LIN {X 0,Y 584.047,Z 358.292,A -85,B 0,C 180,E1 26461.667,E2 26461.667} C_VEL
LIN {X 0,Y 584.039,Z 358.291,A -85,B 0,C 180,E1 26458.43,E2 26458.43} C_VEL
LIN {X 0,Y 584.051,Z 358.293,A -85,B 0,C 180,E1 26455.483,E2 26455.483} C_VEL
LIN {X 0,Y 584.043,Z 358.289,A -85,B 0,C 180,E1 26452.227,E2 26452.227} C_VEL
LIN {X 0,Y 584.062,Z 358.294,A -85,B 0,C 180,E1 26449.245,E2 26449.245} C_VEL
LIN {X 0,Y 584.1,Z 358.29,A -85,B 0,C 180,E1 26446.657,E2 26446.657} C_VEL
LIN {X 0,Y 583.09,Z 358.412,A -85,B 0,C 180,E1 26445.901,E2 26445.901} C_VEL
LIN {X 0,Y 576.621,Z 359.216,A -85,B 0,C 180,E1 26443.781,E2 26443.781} C_VEL
LIN {X 0,Y 576.114,Z 359.282,A -85,B 0,C 180,E1 26443.229,E2 26443.229} C_VEL
LIN {X 0,Y 576.112,Z 359.279,A -85,B 0,C 180,E1 26439.856,E2 26439.856} C_VEL
LIN {X 0,Y 576.152,Z 359.283,A -85,B 0,C 180,E1 26436.692,E2 26436.692} C_VEL
LIN {X 0,Y 576.109,Z 359.279,A -85,B 0,C 180,E1 26433.51,E2 26433.51} C_VEL
LIN {X 0,Y 576.163,Z 359.281,A -85,B 0,C 180,E1 26430.357,E2 26430.357} C_VEL
LIN {X 0,Y 576.11,Z 359.279,A -85,B 0,C 180,E1 26427.131,E2 26427.131} C_VEL
LIN {X 0,Y 576.16,Z 359.278,A -85,B 0,C 180,E1 26423.96,E2 26423.96} C_VEL
LIN {X 0,Y 576.115,Z 359.279,A -85,B 0,C 180,E1 26420.822,E2 26420.822} C_VEL
LIN {X 0,Y 576.152,Z 359.275,A -85,B 0,C 180,E1 26417.54,E2 26417.54} C_VEL
LIN {X 0,Y 576.133,Z 359.281,A -85,B 0,C 180,E1 26414.355,E2 26414.355} C_VEL
LIN {X 0,Y 576.129,Z 359.276,A -85,B 0,C 180,E1 26410.98,E2 26410.98} C_VEL
LIN {X 0,Y 576.156,Z 359.281,A -85,B 0,C 180,E1 26407.772,E2 26407.772} C_VEL
LIN {X 0,Y 576.125,Z 359.275,A -85,B 0,C 180,E1 26404.571,E2 26404.571} C_VEL
LIN {X 0,Y 576.154,Z 359.278,A -85,B 0,C 180,E1 26401.369,E2 26401.369} C_VEL
LIN {X 0,Y 576.129,Z 359.275,A -85,B 0,C 180,E1 26398.16,E2 26398.16} C_VEL
LIN {X 0,Y 576.155,Z 359.27,A -85,B 0,C 180,E1 26394.821,E2 26394.821} C_VEL
LIN {X 0,Y 576.16,Z 359.275,A -85,B 0,C 180,E1 26391.475,E2 26391.475} C_VEL
LIN {X 0,Y 576.135,Z 359.276,A -85,B 0,C 180,E1 26388.199,E2 26388.199} C_VEL
LIN {X 0,Y 576.149,Z 359.283,A -85,B 0,C 180,E1 26384.982,E2 26384.982} C_VEL
LIN {X 0,Y 576.161,Z 359.453,A -85,B 0,C 180,E1 26381.921,E2 26381.921} C_VEL
LIN {X 0,Y 577.208,Z 362.341,A -85,B 0,C 180,E1 26381.665,E2 26381.665} C_VEL
LIN {X 0,Y 582.648,Z 371.022,A -85,B 0,C 180,E1 26381.087,E2 26381.087} C_VEL
LIN {X 0,Y 581.66,Z 578.825,A -85,B 0,C 180,E1 26377.993,E2 26377.993} C_VEL
LIN {X 0,Y 581.046,Z 710.551,A -85,B 0,C 180,E1 26376.056,E2 26376.056} C_VEL
LIN {X 0,Y 580.715,Z 734.129,A -85,B 0,C 180,E1 26375.517,E2 26375.517} C_VEL
LIN {X 0,Y 580.401,Z 756.068,A -85,B 0,C 180,E1 26374.833,E2 26374.833} C_VEL
LIN {X 0,Y 579.918,Z 778.158,A -85,B 0,C 180,E1 26373.951,E2 26373.951} C_VEL
LIN {X 0,Y 579.481,Z 800.389,A -85,B 0,C 180,E1 26372.865,E2 26372.865} C_VEL
LIN {X 0,Y 578.947,Z 821.449,A -85,B 0,C 180,E1 26371.63,E2 26371.63} C_VEL
LIN {X 0,Y 578.423,Z 842.935,A -85,B 0,C 180,E1 26370.146,E2 26370.146} C_VEL
LIN {X 0,Y 577.968,Z 862.118,A -85,B 0,C 180,E1 26368.609,E2 26368.609} C_VEL
LIN {X 0,Y 577.481,Z 880.371,A -85,B 0,C 180,E1 26366.92,E2 26366.92} C_VEL
LIN {X 0,Y 577.086,Z 898.241,A -85,B 0,C 180,E1 26365.027,E2 26365.027} C_VEL
LIN {X 0,Y 576.768,Z 913.925,A -85,B 0,C 180,E1 26363.127,E2 26363.127} C_VEL
LIN {X 0,Y 576.482,Z 927.611,A -85,B 0,C 180,E1 26361.218,E2 26361.218} C_VEL
LIN {X 0,Y 576.279,Z 940.902,A -85,B 0,C 180,E1 26359.096,E2 26359.096} C_VEL
LIN {X 0,Y 576.134,Z 951.802,A -85,B 0,C 180,E1 26357.061,E2 26357.061} C_VEL
LIN {X 0,Y 576.034,Z 962.063,A -85,B 0,C 180,E1 26354.803,E2 26354.803} C_VEL
LIN {X 0,Y 575.951,Z 969.516,A -85,B 0,C 180,E1 26352.833,E2 26352.833} C_VEL
LIN {X 0,Y 575.908,Z 976.629,A -85,B 0,C 180,E1 26350.516,E2 26350.516} C_VEL
LIN {X 0,Y 575.923,Z 981.54,A -85,B 0,C 180,E1 26348.402,E2 26348.402} C_VEL
LIN {X 0,Y 575.899,Z 985.41,A -85,B 0,C 180,E1 26346.027,E2 26346.027} C_VEL
LIN {X 0,Y 575.883,Z 987.332,A -85,B 0,C 180,E1 26343.941,E2 26343.941} C_VEL
LIN {X 0,Y 575.901,Z 987.929,A -85,B 0,C 180,E1 26341.592,E2 26341.592} C_VEL
LIN {X 0,Y 575.91,Z 986.963,A -85,B 0,C 180,E1 26339.421,E2 26339.421} C_VEL
LIN {X 0,Y 575.903,Z 984.298,A -85,B 0,C 180,E1 26337.081,E2 26337.081} C_VEL
LIN {X 0,Y 575.926,Z 980.083,A -85,B 0,C 180,E1 26334.802,E2 26334.802} C_VEL
LIN {X 0,Y 575.937,Z 973.943,A -85,B 0,C 180,E1 26332.455,E2 26332.455} C_VEL
LIN {X 0,Y 576.001,Z 967.203,A -85,B 0,C 180,E1 26330.42,E2 26330.42} C_VEL
LIN {X 0,Y 576.072,Z 958.165,A -85,B 0,C 180,E1 26328.201,E2 26328.201} C_VEL
LIN {X 0,Y 576.199,Z 947.718,A -85,B 0,C 180,E1 26326.042,E2 26326.042} C_VEL
LIN {X 0,Y 576.354,Z 935.657,A -85,B 0,C 180,E1 26323.942,E2 26323.942} C_VEL
LIN {X 0,Y 576.619,Z 922.062,A -85,B 0,C 180,E1 26321.882,E2 26321.882} C_VEL
LIN {X 0,Y 576.933,Z 906.451,A -85,B 0,C 180,E1 26319.846,E2 26319.846} C_VEL
LIN {X 0,Y 577.278,Z 889.678,A -85,B 0,C 180,E1 26317.943,E2 26317.943} C_VEL
LIN {X 0,Y 577.706,Z 871.832,A -85,B 0,C 180,E1 26316.17,E2 26316.17} C_VEL
LIN {X 0,Y 578.182,Z 853.165,A -85,B 0,C 180,E1 26314.557,E2 26314.557} C_VEL
LIN {X 0,Y 578.662,Z 832.887,A -85,B 0,C 180,E1 26313.041,E2 26313.041} C_VEL
LIN {X 0,Y 579.219,Z 811.589,A -85,B 0,C 180,E1 26311.675,E2 26311.675} C_VEL
LIN {X 0,Y 579.672,Z 790.373,A -85,B 0,C 180,E1 26310.529,E2 26310.529} C_VEL
LIN {X 0,Y 580.158,Z 768.038,A -85,B 0,C 180,E1 26309.532,E2 26309.532} C_VEL
LIN {X 0,Y 580.516,Z 746.553,A -85,B 0,C 180,E1 26308.758,E2 26308.758} C_VEL
LIN {X 0,Y 580.89,Z 723.232,A -85,B 0,C 180,E1 26308.119,E2 26308.119} C_VEL
LIN {X 0,Y 581.099,Z 700.855,A -85,B 0,C 180,E1 26307.69,E2 26307.69} C_VEL
LIN {X 0,Y 582.078,Z 488.35,A -85,B 0,C 180,E1 26304.584,E2 26304.584} C_VEL
LIN {X 0,Y 582.542,Z 370.805,A -85,B 0,C 180,E1 26302.811,E2 26302.811} C_VEL
LIN {X 0,Y 576.646,Z 361.193,A -85,B 0,C 180,E1 26302.156,E2 26302.156} C_VEL
LIN {X 0,Y 576.178,Z 359.428,A -85,B 0,C 180,E1 26301.934,E2 26301.934} C_VEL
LIN {X 0,Y 576.126,Z 359.253,A -85,B 0,C 180,E1 26298.728,E2 26298.728} C_VEL
LIN {X 0,Y 576.152,Z 359.274,A -85,B 0,C 180,E1 26295.398,E2 26295.398} C_VEL
LIN {X 0,Y 576.155,Z 359.281,A -85,B 0,C 180,E1 26292.122,E2 26292.122} C_VEL
LIN {X 0,Y 576.139,Z 359.277,A -85,B 0,C 180,E1 26288.886,E2 26288.886} C_VEL
LIN {X 0,Y 576.143,Z 359.277,A -85,B 0,C 180,E1 26285.677,E2 26285.677} C_VEL
LIN {X 0,Y 576.148,Z 359.28,A -85,B 0,C 180,E1 26282.387,E2 26282.387} C_VEL
LIN {X 0,Y 576.156,Z 359.274,A -85,B 0,C 180,E1 26279.006,E2 26279.006} C_VEL
LIN {X 0,Y 576.138,Z 359.281,A -85,B 0,C 180,E1 26275.721,E2 26275.721} C_VEL
LIN {X 0,Y 576.153,Z 359.278,A -85,B 0,C 180,E1 26272.422,E2 26272.422} C_VEL
LIN {X 0,Y 576.123,Z 359.278,A -85,B 0,C 180,E1 26269.197,E2 26269.197} C_VEL
LIN {X 0,Y 576.159,Z 359.283,A -85,B 0,C 180,E1 26265.939,E2 26265.939} C_VEL
LIN {X 0,Y 576.139,Z 359.276,A -85,B 0,C 180,E1 26262.633,E2 26262.633} C_VEL
LIN {X 0,Y 576.113,Z 359.28,A -85,B 0,C 180,E1 26259.303,E2 26259.303} C_VEL
LIN {X 0,Y 576.162,Z 359.277,A -85,B 0,C 180,E1 26256.143,E2 26256.143} C_VEL
LIN {X 0,Y 576.097,Z 359.281,A -85,B 0,C 180,E1 26252.919,E2 26252.919} C_VEL
LIN {X 0,Y 576.163,Z 359.281,A -85,B 0,C 180,E1 26249.785,E2 26249.785} C_VEL
LIN {X 0,Y 576.085,Z 359.283,A -85,B 0,C 180,E1 26246.74,E2 26246.74} C_VEL
LIN {X 0,Y 576.141,Z 359.283,A -85,B 0,C 180,E1 26243.593,E2 26243.593} C_VEL
LIN {X 0,Y 576.074,Z 359.286,A -85,B 0,C 180,E1 26240.562,E2 26240.562} C_VEL
LIN {X 0,Y 576.129,Z 359.285,A -85,B 0,C 180,E1 26237.38,E2 26237.38} C_VEL
LIN {X 0,Y 576.082,Z 359.287,A -85,B 0,C 180,E1 26234.351,E2 26234.351} C_VEL
LIN {X 0,Y 576.127,Z 359.53,A -85,B 0,C 180,E1 26232.179,E2 26232.179} C_VEL
LIN {X 0,Y 577.584,Z 362.943,A -85,B 0,C 180,E1 26231.746,E2 26231.746} C_VEL
LIN {X 0,Y 581.448,Z 371.697,A -85,B 0,C 180,E1 26230.768,E2 26230.768} C_VEL
LIN {X 0,Y 581.237,Z 391.482,A -85,B 0,C 180,E1 26229.398,E2 26229.398} C_VEL
LIN {X 0,Y 582.66,Z 399.109,A -85,B 0,C 180,E1 26229.161,E2 26229.161} C_VEL
LIN {X 0,Y 581.675,Z 605.405,A -85,B 0,C 180,E1 26226.088,E2 26226.088} C_VEL
LIN {X 0,Y 581.041,Z 739.762,A -85,B 0,C 180,E1 26224.113,E2 26224.113} C_VEL
LIN {X 0,Y 580.713,Z 763.529,A -85,B 0,C 180,E1 26223.577,E2 26223.577} C_VEL
LIN {X 0,Y 580.42,Z 784.648,A -85,B 0,C 180,E1 26222.926,E2 26222.926} C_VEL
LIN {X 0,Y 579.923,Z 807.636,A -85,B 0,C 180,E1 26222.019,E2 26222.019} C_VEL
LIN {X 0,Y 579.517,Z 829.395,A -85,B 0,C 180,E1 26220.965,E2 26220.965} C_VEL
LIN {X 0,Y 578.968,Z 849.896,A -85,B 0,C 180,E1 26219.771,E2 26219.771} C_VEL
LIN {X 0,Y 578.482,Z 871.118,A -85,B 0,C 180,E1 26218.326,E2 26218.326} C_VEL
LIN {X 0,Y 577.997,Z 889.882,A -85,B 0,C 180,E1 26216.842,E2 26216.842} C_VEL
LIN {X 0,Y 577.555,Z 907.881,A -85,B 0,C 180,E1 26215.208,E2 26215.208} C_VEL
LIN {X 0,Y 577.191,Z 924.959,A -85,B 0,C 180,E1 26213.448,E2 26213.448} C_VEL
LIN {X 0,Y 576.817,Z 940.825,A -85,B 0,C 180,E1 26211.563,E2 26211.563} C_VEL
LIN {X 0,Y 576.519,Z 956.316,A -85,B 0,C 180,E1 26209.452,E2 26209.452} C_VEL
LIN {X 0,Y 576.322,Z 969.346,A -85,B 0,C 180,E1 26207.411,E2 26207.411} C_VEL
LIN {X 0,Y 576.149,Z 980.824,A -85,B 0,C 180,E1 26205.297,E2 26205.297} C_VEL
LIN {X 0,Y 576.037,Z 990.869,A -85,B 0,C 180,E1 26203.146,E2 26203.146} C_VEL
LIN {X 0,Y 575.953,Z 999.042,A -85,B 0,C 180,E1 26201.011,E2 26201.011} C_VEL
LIN {X 0,Y 575.942,Z 1005.767,A -85,B 0,C 180,E1 26198.891,E2 26198.891} C_VEL
LIN {X 0,Y 575.907,Z 1011.041,A -85,B 0,C 180,E1 26196.683,E2 26196.683} C_VEL
LIN {X 0,Y 575.902,Z 1014.908,A -85,B 0,C 180,E1 26194.484,E2 26194.484} C_VEL
LIN {X 0,Y 575.915,Z 1017.187,A -85,B 0,C 180,E1 26192.192,E2 26192.192} C_VEL
LIN {X 0,Y 575.908,Z 1017.985,A -85,B 0,C 180,E1 26189.904,E2 26189.904} C_VEL
LIN {X 0,Y 575.915,Z 1017.124,A -85,B 0,C 180,E1 26187.715,E2 26187.715} C_VEL
LIN {X 0,Y 575.901,Z 1014.759,A -85,B 0,C 180,E1 26185.422,E2 26185.422} C_VEL
LIN {X 0,Y 575.908,Z 1011.054,A -85,B 0,C 180,E1 26183.323,E2 26183.323} C_VEL
LIN {X 0,Y 575.945,Z 1005.56,A -85,B 0,C 180,E1 26181.039,E2 26181.039} C_VEL
LIN {X 0,Y 575.955,Z 998.707,A -85,B 0,C 180,E1 26178.893,E2 26178.893} C_VEL
LIN {X 0,Y 576.039,Z 990.472,A -85,B 0,C 180,E1 26176.758,E2 26176.758} C_VEL
LIN {X 0,Y 576.149,Z 980.857,A -85,B 0,C 180,E1 26174.709,E2 26174.709} C_VEL
LIN {X 0,Y 576.324,Z 969.344,A -85,B 0,C 180,E1 26172.589,E2 26172.589} C_VEL
LIN {X 0,Y 576.518,Z 956.359,A -85,B 0,C 180,E1 26170.554,E2 26170.554} C_VEL
LIN {X 0,Y 576.814,Z 940.877,A -85,B 0,C 180,E1 26168.444,E2 26168.444} C_VEL
LIN {X 0,Y 577.197,Z 924.713,A -85,B 0,C 180,E1 26166.525,E2 26166.525} C_VEL
LIN {X 0,Y 577.572,Z 907.396,A -85,B 0,C 180,E1 26164.744,E2 26164.744} C_VEL
LIN {X 0,Y 578.017,Z 888.638,A -85,B 0,C 180,E1 26163.055,E2 26163.055} C_VEL
LIN {X 0,Y 578.526,Z 869.809,A -85,B 0,C 180,E1 26161.576,E2 26161.576} C_VEL
LIN {X 0,Y 578.991,Z 849.113,A -85,B 0,C 180,E1 26160.18,E2 26160.18} C_VEL
LIN {X 0,Y 579.542,Z 827.764,A -85,B 0,C 180,E1 26158.95,E2 26158.95} C_VEL
LIN {X 0,Y 579.95,Z 806.518,A -85,B 0,C 180,E1 26157.932,E2 26157.932} C_VEL
LIN {X 0,Y 580.431,Z 783.297,A -85,B 0,C 180,E1 26157.029,E2 26157.029} C_VEL
LIN {X 0,Y 580.725,Z 762.511,A -85,B 0,C 180,E1 26156.395,E2 26156.395} C_VEL
LIN {X 0,Y 581.045,Z 738.852,A -85,B 0,C 180,E1 26155.872,E2 26155.872} C_VEL
LIN {X 0,Y 582.084,Z 515.398,A -85,B 0,C 180,E1 26152.584,E2 26152.584} C_VEL
LIN {X 0,Y 582.507,Z 397.407,A -85,B 0,C 180,E1 26150.8,E2 26150.8} C_VEL
LIN {X 0,Y 581.157,Z 390.898,A -85,B 0,C 180,E1 26150.577,E2 26150.577} C_VEL
LIN {X 0,Y 581.327,Z 371.135,A -85,B 0,C 180,E1 26149.181,E2 26149.181} C_VEL
LIN {X 0,Y 577.109,Z 362.215,A -85,B 0,C 180,E1 26148.157,E2 26148.157} C_VEL
LIN {X 0,Y 576.112,Z 359.423,A -85,B 0,C 180,E1 26147.795,E2 26147.795} C_VEL
LIN {X 0,Y 576.105,Z 359.274,A -85,B 0,C 180,E1 26144.926,E2 26144.926} C_VEL
LIN {X 0,Y 576.089,Z 359.285,A -85,B 0,C 180,E1 26141.586,E2 26141.586} C_VEL
LIN {X 0,Y 576.108,Z 359.277,A -85,B 0,C 180,E1 26138.656,E2 26138.656} C_VEL
LIN {X 0,Y 576.083,Z 359.275,A -85,B 0,C 180,E1 26135.429,E2 26135.429} C_VEL
LIN {X 0,Y 576.097,Z 359.284,A -85,B 0,C 180,E1 26132.549,E2 26132.549} C_VEL
LIN {X 0,Y 576.081,Z 359.282,A -85,B 0,C 180,E1 26129.304,E2 26129.304} C_VEL
LIN {X 0,Y 576.083,Z 359.284,A -85,B 0,C 180,E1 26126.49,E2 26126.49} C_VEL
LIN {X 0,Y 576.079,Z 359.283,A -85,B 0,C 180,E1 26123.094,E2 26123.094} C_VEL
LIN {X 0,Y 576.094,Z 359.283,A -85,B 0,C 180,E1 26120.205,E2 26120.205} C_VEL
LIN {X 0,Y 576.086,Z 359.283,A -85,B 0,C 180,E1 26116.952,E2 26116.952} C_VEL
LIN {X 0,Y 576.097,Z 359.282,A -85,B 0,C 180,E1 26114.048,E2 26114.048} C_VEL
LIN {X 0,Y 576.087,Z 359.282,A -85,B 0,C 180,E1 26110.702,E2 26110.702} C_VEL
LIN {X 0,Y 576.114,Z 359.281,A -85,B 0,C 180,E1 26107.74,E2 26107.74} C_VEL
LIN {X 0,Y 576.09,Z 359.281,A -85,B 0,C 180,E1 26104.479,E2 26104.479} C_VEL
LIN {X 0,Y 576.128,Z 359.281,A -85,B 0,C 180,E1 26101.491,E2 26101.491} C_VEL
LIN {X 0,Y 576.094,Z 359.28,A -85,B 0,C 180,E1 26098.309,E2 26098.309} C_VEL
LIN {X 0,Y 576.141,Z 359.282,A -85,B 0,C 180,E1 26095.221,E2 26095.221} C_VEL
LIN {X 0,Y 576.095,Z 359.278,A -85,B 0,C 180,E1 26092.018,E2 26092.018} C_VEL
LIN {X 0,Y 576.16,Z 359.28,A -85,B 0,C 180,E1 26088.893,E2 26088.893} C_VEL
LIN {X 0,Y 576.098,Z 359.28,A -85,B 0,C 180,E1 26085.732,E2 26085.732} C_VEL
LIN {X 0,Y 576.114,Z 359.282,A -85,B 0,C 180,E1 26083.229,E2 26083.229} C_VEL
LIN {X 0,Y 575.164,Z 359.406,A -85,B 0,C 180,E1 26082.463,E2 26082.463} C_VEL
LIN {X 0,Y 568.626,Z 360.216,A -85,B 0,C 180,E1 26080.257,E2 26080.257} C_VEL
LIN {X 0,Y 568.168,Z 360.268,A -85,B 0,C 180,E1 26079.752,E2 26079.752} C_VEL
LIN {X 0,Y 568.222,Z 360.271,A -85,B 0,C 180,E1 26076.567,E2 26076.567} C_VEL
LIN {X 0,Y 568.167,Z 360.269,A -85,B 0,C 180,E1 26073.336,E2 26073.336} C_VEL
LIN {X 0,Y 568.223,Z 360.266,A -85,B 0,C 180,E1 26070.134,E2 26070.134} C_VEL
LIN {X 0,Y 568.176,Z 360.27,A -85,B 0,C 180,E1 26066.884,E2 26066.884} C_VEL
LIN {X 0,Y 568.193,Z 360.266,A -85,B 0,C 180,E1 26063.502,E2 26063.502} C_VEL
LIN {X 0,Y 568.219,Z 360.272,A -85,B 0,C 180,E1 26060.253,E2 26060.253} C_VEL
LIN {X 0,Y 568.178,Z 360.268,A -85,B 0,C 180,E1 26056.905,E2 26056.905} C_VEL
LIN {X 0,Y 568.219,Z 360.264,A -85,B 0,C 180,E1 26053.679,E2 26053.679} C_VEL
LIN {X 0,Y 568.184,Z 360.269,A -85,B 0,C 180,E1 26050.486,E2 26050.486} C_VEL
LIN {X 0,Y 568.21,Z 360.264,A -85,B 0,C 180,E1 26047.12,E2 26047.12} C_VEL
LIN {X 0,Y 568.217,Z 360.262,A -85,B 0,C 180,E1 26043.778,E2 26043.778} C_VEL
LIN {X 0,Y 568.187,Z 360.267,A -85,B 0,C 180,E1 26040.427,E2 26040.427} C_VEL
LIN {X 0,Y 568.215,Z 360.267,A -85,B 0,C 180,E1 26037.222,E2 26037.222} C_VEL
LIN {X 0,Y 568.193,Z 360.264,A -85,B 0,C 180,E1 26033.98,E2 26033.98} C_VEL
LIN {X 0,Y 568.215,Z 360.261,A -85,B 0,C 180,E1 26030.601,E2 26030.601} C_VEL
LIN {X 0,Y 568.214,Z 360.247,A -85,B 0,C 180,E1 26027.296,E2 26027.296} C_VEL
LIN {X 0,Y 568.197,Z 360.263,A -85,B 0,C 180,E1 26024.05,E2 26024.05} C_VEL
LIN {X 0,Y 568.236,Z 360.408,A -85,B 0,C 180,E1 26022.573,E2 26022.573} C_VEL
LIN {X 0,Y 568.508,Z 361.583,A -85,B 0,C 180,E1 26022.412,E2 26022.412} C_VEL
LIN {X 0,Y 570.42,Z 364.804,A -85,B 0,C 180,E1 26022.194,E2 26022.194} C_VEL
LIN {X 0,Y 576.42,Z 374.475,A -85,B 0,C 180,E1 26021.538,E2 26021.538} C_VEL
LIN {X 0,Y 575.163,Z 582.912,A -85,B 0,C 180,E1 26018.403,E2 26018.403} C_VEL
LIN {X 0,Y 574.411,Z 710.911,A -85,B 0,C 180,E1 26016.5,E2 26016.5} C_VEL
LIN {X 0,Y 573.996,Z 734.544,A -85,B 0,C 180,E1 26015.952,E2 26015.952} C_VEL
LIN {X 0,Y 573.592,Z 756.803,A -85,B 0,C 180,E1 26015.248,E2 26015.248} C_VEL
LIN {X 0,Y 572.992,Z 778.919,A -85,B 0,C 180,E1 26014.35,E2 26014.35} C_VEL
LIN {X 0,Y 572.429,Z 801.045,A -85,B 0,C 180,E1 26013.251,E2 26013.251} C_VEL
LIN {X 0,Y 571.766,Z 822.066,A -85,B 0,C 180,E1 26012.001,E2 26012.001} C_VEL
LIN {X 0,Y 571.111,Z 843.462,A -85,B 0,C 180,E1 26010.498,E2 26010.498} C_VEL
LIN {X 0,Y 570.524,Z 862.609,A -85,B 0,C 180,E1 26008.943,E2 26008.943} C_VEL
LIN {X 0,Y 569.927,Z 880.796,A -85,B 0,C 180,E1 26007.232,E2 26007.232} C_VEL
LIN {X 0,Y 569.43,Z 898.173,A -85,B 0,C 180,E1 26005.364,E2 26005.364} C_VEL
LIN {X 0,Y 569.01,Z 913.859,A -85,B 0,C 180,E1 26003.439,E2 26003.439} C_VEL
LIN {X 0,Y 568.646,Z 928.228,A -85,B 0,C 180,E1 26001.402,E2 26001.402} C_VEL
LIN {X 0,Y 568.383,Z 941.407,A -85,B 0,C 180,E1 25999.251,E2 25999.251} C_VEL
LIN {X 0,Y 568.195,Z 952.527,A -85,B 0,C 180,E1 25997.132,E2 25997.132} C_VEL
LIN {X 0,Y 568.068,Z 962.412,A -85,B 0,C 180,E1 25994.898,E2 25994.898} C_VEL
LIN {X 0,Y 567.968,Z 970.185,A -85,B 0,C 180,E1 25992.795,E2 25992.795} C_VEL
LIN {X 0,Y 567.911,Z 977.088,A -85,B 0,C 180,E1 25990.455,E2 25990.455} C_VEL
LIN {X 0,Y 567.916,Z 981.939,A -85,B 0,C 180,E1 25988.299,E2 25988.299} C_VEL
LIN {X 0,Y 567.91,Z 985.63,A -85,B 0,C 180,E1 25985.89,E2 25985.89} C_VEL
LIN {X 0,Y 567.884,Z 987.466,A -85,B 0,C 180,E1 25983.771,E2 25983.771} C_VEL
LIN {X 0,Y 567.903,Z 987.885,A -85,B 0,C 180,E1 25981.385,E2 25981.385} C_VEL
LIN {X 0,Y 567.918,Z 986.827,A -85,B 0,C 180,E1 25979.179,E2 25979.179} C_VEL
LIN {X 0,Y 567.917,Z 983.966,A -85,B 0,C 180,E1 25976.8,E2 25976.8} C_VEL
LIN {X 0,Y 567.933,Z 979.606,A -85,B 0,C 180,E1 25974.479,E2 25974.479} C_VEL
LIN {X 0,Y 567.942,Z 973.637,A -85,B 0,C 180,E1 25972.216,E2 25972.216} C_VEL
LIN {X 0,Y 568.014,Z 966.205,A -85,B 0,C 180,E1 25969.971,E2 25969.971} C_VEL
LIN {X 0,Y 568.127,Z 957.301,A -85,B 0,C 180,E1 25967.811,E2 25967.811} C_VEL
LIN {X 0,Y 568.31,Z 946.33,A -85,B 0,C 180,E1 25965.553,E2 25965.553} C_VEL
LIN {X 0,Y 568.536,Z 934.047,A -85,B 0,C 180,E1 25963.419,E2 25963.419} C_VEL
LIN {X 0,Y 568.864,Z 919.438,A -85,B 0,C 180,E1 25961.233,E2 25961.233} C_VEL
LIN {X 0,Y 569.285,Z 903.948,A -85,B 0,C 180,E1 25959.219,E2 25959.219} C_VEL
LIN {X 0,Y 569.763,Z 887.305,A -85,B 0,C 180,E1 25957.347,E2 25957.347} C_VEL
LIN {X 0,Y 570.29,Z 869.121,A -85,B 0,C 180,E1 25955.558,E2 25955.558} C_VEL
LIN {X 0,Y 570.897,Z 850.628,A -85,B 0,C 180,E1 25953.966,E2 25953.966} C_VEL
LIN {X 0,Y 571.518,Z 830.685,A -85,B 0,C 180,E1 25952.486,E2 25952.486} C_VEL
LIN {X 0,Y 572.168,Z 808.837,A -85,B 0,C 180,E1 25951.097,E2 25951.097} C_VEL
LIN {X 0,Y 572.796,Z 787.97,A -85,B 0,C 180,E1 25949.984,E2 25949.984} C_VEL
LIN {X 0,Y 573.326,Z 765.683,A -85,B 0,C 180,E1 25949.001,E2 25949.001} C_VEL
LIN {X 0,Y 573.876,Z 743.3,A -85,B 0,C 180,E1 25948.21,E2 25948.21} C_VEL
LIN {X 0,Y 574.238,Z 720.543,A -85,B 0,C 180,E1 25947.61,E2 25947.61} C_VEL
LIN {X 0,Y 574.534,Z 696.509,A -85,B 0,C 180,E1 25947.173,E2 25947.173} C_VEL
LIN {X 0,Y 575.749,Z 483.143,A -85,B 0,C 180,E1 25944.02,E2 25944.02} C_VEL
LIN {X 0,Y 576.263,Z 374.074,A -85,B 0,C 180,E1 25942.353,E2 25942.353} C_VEL
LIN {X 0,Y 570.255,Z 364.674,A -85,B 0,C 180,E1 25941.7,E2 25941.7} C_VEL
LIN {X 0,Y 568.449,Z 361.484,A -85,B 0,C 180,E1 25941.488,E2 25941.488} C_VEL
LIN {X 0,Y 568.198,Z 360.347,A -85,B 0,C 180,E1 25941.292,E2 25941.292} C_VEL
LIN {X 0,Y 568.214,Z 360.243,A -85,B 0,C 180,E1 25938.041,E2 25938.041} C_VEL
LIN {X 0,Y 568.19,Z 360.263,A -85,B 0,C 180,E1 25934.783,E2 25934.783} C_VEL
LIN {X 0,Y 568.219,Z 360.264,A -85,B 0,C 180,E1 25931.44,E2 25931.44} C_VEL
LIN {X 0,Y 568.218,Z 360.269,A -85,B 0,C 180,E1 25928.093,E2 25928.093} C_VEL
LIN {X 0,Y 568.203,Z 360.265,A -85,B 0,C 180,E1 25924.744,E2 25924.744} C_VEL
LIN {X 0,Y 568.201,Z 360.267,A -85,B 0,C 180,E1 25921.513,E2 25921.513} C_VEL
LIN {X 0,Y 568.213,Z 360.27,A -85,B 0,C 180,E1 25918.286,E2 25918.286} C_VEL
LIN {X 0,Y 568.211,Z 360.263,A -85,B 0,C 180,E1 25914.953,E2 25914.953} C_VEL
LIN {X 0,Y 568.193,Z 360.27,A -85,B 0,C 180,E1 25911.602,E2 25911.602} C_VEL
LIN {X 0,Y 568.218,Z 360.267,A -85,B 0,C 180,E1 25908.326,E2 25908.326} C_VEL
LIN {X 0,Y 568.179,Z 360.268,A -85,B 0,C 180,E1 25905.113,E2 25905.113} C_VEL
LIN {X 0,Y 568.214,Z 360.272,A -85,B 0,C 180,E1 25901.847,E2 25901.847} C_VEL
LIN {X 0,Y 568.186,Z 360.266,A -85,B 0,C 180,E1 25898.638,E2 25898.638} C_VEL
LIN {X 0,Y 568.173,Z 360.272,A -85,B 0,C 180,E1 25895.351,E2 25895.351} C_VEL
LIN {X 0,Y 568.205,Z 360.268,A -85,B 0,C 180,E1 25892.205,E2 25892.205} C_VEL
LIN {X 0,Y 568.151,Z 360.272,A -85,B 0,C 180,E1 25888.961,E2 25888.961} C_VEL
LIN {X 0,Y 568.223,Z 360.269,A -85,B 0,C 180,E1 25885.796,E2 25885.796} C_VEL
LIN {X 0,Y 568.139,Z 360.274,A -85,B 0,C 180,E1 25882.616,E2 25882.616} C_VEL
LIN {X 0,Y 568.195,Z 360.272,A -85,B 0,C 180,E1 25879.483,E2 25879.483} C_VEL
LIN {X 0,Y 568.142,Z 360.277,A -85,B 0,C 180,E1 25876.33,E2 25876.33} C_VEL
LIN {X 0,Y 568.167,Z 360.246,A -85,B 0,C 180,E1 25873.065,E2 25873.065} C_VEL
LIN {X 0,Y 568.222,Z 360.733,A -85,B 0,C 180,E1 25872.784,E2 25872.784} C_VEL
LIN {X 0,Y 574.864,Z 375.383,A -85,B 0,C 180,E1 25871.064,E2 25871.064} C_VEL
LIN {X 0,Y 574.653,Z 391.507,A -85,B 0,C 180,E1 25869.939,E2 25869.939} C_VEL
LIN {X 0,Y 576.441,Z 400.829,A -85,B 0,C 180,E1 25869.639,E2 25869.639} C_VEL
LIN {X 0,Y 575.197,Z 607.147,A -85,B 0,C 180,E1 25866.533,E2 25866.533} C_VEL
LIN {X 0,Y 574.407,Z 739.87,A -85,B 0,C 180,E1 25864.56,E2 25864.56} C_VEL
LIN {X 0,Y 573.995,Z 763.685,A -85,B 0,C 180,E1 25864.019,E2 25864.019} C_VEL
LIN {X 0,Y 573.619,Z 785.243,A -85,B 0,C 180,E1 25863.346,E2 25863.346} C_VEL
LIN {X 0,Y 573.022,Z 807.638,A -85,B 0,C 180,E1 25862.451,E2 25862.451} C_VEL
LIN {X 0,Y 572.504,Z 828.746,A -85,B 0,C 180,E1 25861.423,E2 25861.423} C_VEL
LIN {X 0,Y 571.828,Z 849.899,A -85,B 0,C 180,E1 25860.181,E2 25860.181} C_VEL
LIN {X 0,Y 571.196,Z 871.115,A -85,B 0,C 180,E1 25858.72,E2 25858.72} C_VEL
LIN {X 0,Y 570.578,Z 889.884,A -85,B 0,C 180,E1 25857.22,E2 25857.22} C_VEL
LIN {X 0,Y 570.014,Z 908.435,A -85,B 0,C 180,E1 25855.51,E2 25855.51} C_VEL
LIN {X 0,Y 569.525,Z 925.597,A -85,B 0,C 180,E1 25853.708,E2 25853.708} C_VEL
LIN {X 0,Y 569.061,Z 941.675,A -85,B 0,C 180,E1 25851.763,E2 25851.763} C_VEL
LIN {X 0,Y 568.708,Z 956.318,A -85,B 0,C 180,E1 25849.731,E2 25849.731} C_VEL
LIN {X 0,Y 568.446,Z 968.994,A -85,B 0,C 180,E1 25847.718,E2 25847.718} C_VEL
LIN {X 0,Y 568.22,Z 980.305,A -85,B 0,C 180,E1 25845.621,E2 25845.621} C_VEL
LIN {X 0,Y 568.078,Z 989.985,A -85,B 0,C 180,E1 25843.541,E2 25843.541} C_VEL
LIN {X 0,Y 567.984,Z 998.484,A -85,B 0,C 180,E1 25841.329,E2 25841.329} C_VEL
LIN {X 0,Y 567.947,Z 1005.164,A -85,B 0,C 180,E1 25839.221,E2 25839.221} C_VEL
LIN {X 0,Y 567.896,Z 1010.628,A -85,B 0,C 180,E1 25836.981,E2 25836.981} C_VEL
LIN {X 0,Y 567.907,Z 1014.272,A -85,B 0,C 180,E1 25834.952,E2 25834.952} C_VEL
LIN {X 0,Y 567.915,Z 1016.986,A -85,B 0,C 180,E1 25832.526,E2 25832.526} C_VEL
LIN {X 0,Y 567.887,Z 1017.916,A -85,B 0,C 180,E1 25830.407,E2 25830.407} C_VEL
LIN {X 0,Y 567.913,Z 1017.326,A -85,B 0,C 180,E1 25827.985,E2 25827.985} C_VEL
LIN {X 0,Y 567.912,Z 1015.28,A -85,B 0,C 180,E1 25825.763,E2 25825.763} C_VEL
LIN {X 0,Y 567.919,Z 1011.467,A -85,B 0,C 180,E1 25823.432,E2 25823.432} C_VEL
LIN {X 0,Y 567.939,Z 1006.559,A -85,B 0,C 180,E1 25821.295,E2 25821.295} C_VEL
LIN {X 0,Y 567.969,Z 999.776,A -85,B 0,C 180,E1 25819.044,E2 25819.044} C_VEL
LIN {X 0,Y 568.067,Z 992.122,A -85,B 0,C 180,E1 25816.984,E2 25816.984} C_VEL
LIN {X 0,Y 568.21,Z 981.613,A -85,B 0,C 180,E1 25814.642,E2 25814.642} C_VEL
LIN {X 0,Y 568.424,Z 970.259,A -85,B 0,C 180,E1 25812.499,E2 25812.499} C_VEL
LIN {X 0,Y 568.67,Z 957.593,A -85,B 0,C 180,E1 25810.46,E2 25810.46} C_VEL
LIN {X 0,Y 569.028,Z 943.416,A -85,B 0,C 180,E1 25808.459,E2 25808.459} C_VEL
LIN {X 0,Y 569.447,Z 927.936,A -85,B 0,C 180,E1 25806.565,E2 25806.565} C_VEL
LIN {X 0,Y 569.949,Z 910.161,A -85,B 0,C 180,E1 25804.661,E2 25804.661} C_VEL
LIN {X 0,Y 570.534,Z 891.947,A -85,B 0,C 180,E1 25802.954,E2 25802.954} C_VEL
LIN {X 0,Y 571.138,Z 872.671,A -85,B 0,C 180,E1 25801.398,E2 25801.398} C_VEL
LIN {X 0,Y 571.758,Z 852.033,A -85,B 0,C 180,E1 25799.954,E2 25799.954} C_VEL
LIN {X 0,Y 572.397,Z 831.916,A -85,B 0,C 180,E1 25798.753,E2 25798.753} C_VEL
LIN {X 0,Y 572.972,Z 809.416,A -85,B 0,C 180,E1 25797.628,E2 25797.628} C_VEL
LIN {X 0,Y 573.578,Z 787.495,A -85,B 0,C 180,E1 25796.732,E2 25796.732} C_VEL
LIN {X 0,Y 573.979,Z 765.055,A -85,B 0,C 180,E1 25796.02,E2 25796.02} C_VEL
LIN {X 0,Y 574.39,Z 742.213,A -85,B 0,C 180,E1 25795.48,E2 25795.48} C_VEL
LIN {X 0,Y 574.737,Z 689.171,A -85,B 0,C 180,E1 25794.673,E2 25794.673} C_VEL
LIN {X 0,Y 575.914,Z 482.954,A -85,B 0,C 180,E1 25791.609,E2 25791.609} C_VEL
LIN {X 0,Y 576.292,Z 399.178,A -85,B 0,C 180,E1 25790.323,E2 25790.323} C_VEL
LIN {X 0,Y 574.551,Z 390.636,A -85,B 0,C 180,E1 25790.02,E2 25790.02} C_VEL
LIN {X 0,Y 574.864,Z 375.383,A -85,B 0,C 180,E1 25788.936,E2 25788.936} C_VEL
LIN {X 0,Y 569.72,Z 364.118,A -85,B 0,C 180,E1 25787.633,E2 25787.633} C_VEL
LIN {X 0,Y 568.195,Z 360.554,A -85,B 0,C 180,E1 25787.177,E2 25787.177} C_VEL
LIN {X 0,Y 568.185,Z 360.275,A -85,B 0,C 180,E1 25786.112,E2 25786.112} C_VEL
LIN {X 0,Y 568.149,Z 360.262,A -85,B 0,C 180,E1 25783.092,E2 25783.092} C_VEL
LIN {X 0,Y 568.16,Z 360.263,A -85,B 0,C 180,E1 25779.74,E2 25779.74} C_VEL
LIN {X 0,Y 568.151,Z 360.273,A -85,B 0,C 180,E1 25776.808,E2 25776.808} C_VEL
LIN {X 0,Y 568.146,Z 360.274,A -85,B 0,C 180,E1 25773.424,E2 25773.424} C_VEL
LIN {X 0,Y 568.16,Z 360.264,A -85,B 0,C 180,E1 25770.452,E2 25770.452} C_VEL
LIN {X 0,Y 568.14,Z 360.273,A -85,B 0,C 180,E1 25767.23,E2 25767.23} C_VEL
LIN {X 0,Y 568.157,Z 360.274,A -85,B 0,C 180,E1 25764.286,E2 25764.286} C_VEL
LIN {X 0,Y 568.142,Z 360.272,A -85,B 0,C 180,E1 25761.039,E2 25761.039} C_VEL
LIN {X 0,Y 568.167,Z 360.273,A -85,B 0,C 180,E1 25758.042,E2 25758.042} C_VEL
LIN {X 0,Y 568.143,Z 360.27,A -85,B 0,C 180,E1 25754.784,E2 25754.784} C_VEL
LIN {X 0,Y 568.181,Z 360.272,A -85,B 0,C 180,E1 25751.778,E2 25751.778} C_VEL
LIN {X 0,Y 568.144,Z 360.269,A -85,B 0,C 180,E1 25748.525,E2 25748.525} C_VEL
LIN {X 0,Y 568.204,Z 360.271,A -85,B 0,C 180,E1 25745.452,E2 25745.452} C_VEL
LIN {X 0,Y 568.147,Z 360.268,A -85,B 0,C 180,E1 25742.218,E2 25742.218} C_VEL
LIN {X 0,Y 568.221,Z 360.268,A -85,B 0,C 180,E1 25739.092,E2 25739.092} C_VEL
LIN {X 0,Y 568.151,Z 360.27,A -85,B 0,C 180,E1 25735.963,E2 25735.963} C_VEL
LIN {X 0,Y 568.22,Z 360.266,A -85,B 0,C 180,E1 25732.823,E2 25732.823} C_VEL
LIN {X 0,Y 568.158,Z 360.271,A -85,B 0,C 180,E1 25729.659,E2 25729.659} C_VEL
LIN {X 0,Y 568.21,Z 360.266,A -85,B 0,C 180,E1 25726.465,E2 25726.465} C_VEL
LIN {X 0,Y 568.169,Z 360.271,A -85,B 0,C 180,E1 25723.33,E2 25723.33} C_VEL
LIN {X 0,Y 568.179,Z 360.268,A -85,B 0,C 180,E1 25719.93,E2 25719.93} C_VEL
LIN {X 0,Y 568.168,Z 360.268,A -85,B 0,C 180,E1 25719.752,E2 25719.752} C_VEL
LIN {X 0,Y 567.175,Z 360.399,A -85,B 0,C 180,E1 25718.976,E2 25718.976} C_VEL
LIN {X 0,Y 560.736,Z 361.203,A -85,B 0,C 180,E1 25716.738,E2 25716.738} C_VEL
LIN {X 0,Y 560.28,Z 361.254,A -85,B 0,C 180,E1 25716.227,E2 25716.227} C_VEL
LIN {X 0,Y 560.236,Z 361.259,A -85,B 0,C 180,E1 25713.043,E2 25713.043} C_VEL
LIN {X 0,Y 560.249,Z 361.255,A -85,B 0,C 180,E1 25709.664,E2 25709.664} C_VEL
LIN {X 0,Y 560.274,Z 361.262,A -85,B 0,C 180,E1 25706.411,E2 25706.411} C_VEL
LIN {X 0,Y 560.236,Z 361.257,A -85,B 0,C 180,E1 25703.079,E2 25703.079} C_VEL
LIN {X 0,Y 560.283,Z 361.252,A -85,B 0,C 180,E1 25699.758,E2 25699.758} C_VEL
LIN {X 0,Y 560.256,Z 361.26,A -85,B 0,C 180,E1 25696.426,E2 25696.426} C_VEL
LIN {X 0,Y 560.252,Z 361.252,A -85,B 0,C 180,E1 25693.113,E2 25693.113} C_VEL
LIN {X 0,Y 560.278,Z 361.259,A -85,B 0,C 180,E1 25689.835,E2 25689.835} C_VEL
LIN {X 0,Y 560.245,Z 361.257,A -85,B 0,C 180,E1 25686.572,E2 25686.572} C_VEL
LIN {X 0,Y 560.28,Z 361.25,A -85,B 0,C 180,E1 25683.215,E2 25683.215} C_VEL
LIN {X 0,Y 560.271,Z 361.253,A -85,B 0,C 180,E1 25679.851,E2 25679.851} C_VEL
LIN {X 0,Y 560.256,Z 361.256,A -85,B 0,C 180,E1 25676.493,E2 25676.493} C_VEL
LIN {X 0,Y 560.275,Z 361.258,A -85,B 0,C 180,E1 25673.21,E2 25673.21} C_VEL
LIN {X 0,Y 560.256,Z 361.256,A -85,B 0,C 180,E1 25669.926,E2 25669.926} C_VEL
LIN {X 0,Y 560.278,Z 361.228,A -85,B 0,C 180,E1 25666.587,E2 25666.587} C_VEL
LIN {X 0,Y 560.306,Z 361.432,A -85,B 0,C 180,E1 25663.253,E2 25663.253} C_VEL
LIN {X 0,Y 560.605,Z 362.708,A -85,B 0,C 180,E1 25663.083,E2 25663.083} C_VEL
LIN {X 0,Y 562.536,Z 365.854,A -85,B 0,C 180,E1 25662.86,E2 25662.86} C_VEL
LIN {X 0,Y 563.768,Z 367.591,A -85,B 0,C 180,E1 25662.723,E2 25662.723} C_VEL
LIN {X 0,Y 570.224,Z 377.843,A -85,B 0,C 180,E1 25662,E2 25662} C_VEL
LIN {X 0,Y 568.704,Z 585.941,A -85,B 0,C 180,E1 25658.838,E2 25658.838} C_VEL
LIN {X 0,Y 567.812,Z 711.089,A -85,B 0,C 180,E1 25656.956,E2 25656.956} C_VEL
LIN {X 0,Y 567.317,Z 734.728,A -85,B 0,C 180,E1 25656.403,E2 25656.403} C_VEL
LIN {X 0,Y 566.808,Z 757.694,A -85,B 0,C 180,E1 25655.666,E2 25655.666} C_VEL
LIN {X 0,Y 566.098,Z 779.675,A -85,B 0,C 180,E1 25654.758,E2 25654.758} C_VEL
LIN {X 0,Y 565.403,Z 801.701,A -85,B 0,C 180,E1 25653.647,E2 25653.647} C_VEL
LIN {X 0,Y 564.616,Z 822.678,A -85,B 0,C 180,E1 25652.382,E2 25652.382} C_VEL
LIN {X 0,Y 563.848,Z 843.335,A -85,B 0,C 180,E1 25650.911,E2 25650.911} C_VEL
LIN {X 0,Y 563.11,Z 862.514,A -85,B 0,C 180,E1 25649.336,E2 25649.336} C_VEL
LIN {X 0,Y 562.415,Z 880.672,A -85,B 0,C 180,E1 25647.606,E2 25647.606} C_VEL
LIN {X 0,Y 561.793,Z 898.106,A -85,B 0,C 180,E1 25645.71,E2 25645.71} C_VEL
LIN {X 0,Y 561.267,Z 913.897,A -85,B 0,C 180,E1 25643.744,E2 25643.744} C_VEL
LIN {X 0,Y 560.837,Z 928.296,A -85,B 0,C 180,E1 25641.674,E2 25641.674} C_VEL
LIN {X 0,Y 560.489,Z 941.959,A -85,B 0,C 180,E1 25639.401,E2 25639.401} C_VEL
LIN {X 0,Y 560.256,Z 953.203,A -85,B 0,C 180,E1 25637.212,E2 25637.212} C_VEL
LIN {X 0,Y 560.1,Z 962.88,A -85,B 0,C 180,E1 25634.966,E2 25634.966} C_VEL
LIN {X 0,Y 559.985,Z 970.854,A -85,B 0,C 180,E1 25632.756,E2 25632.756} C_VEL
LIN {X 0,Y 559.918,Z 977.305,A -85,B 0,C 180,E1 25630.49,E2 25630.49} C_VEL
LIN {X 0,Y 559.919,Z 982.115,A -85,B 0,C 180,E1 25628.304,E2 25628.304} C_VEL
LIN {X 0,Y 559.913,Z 985.731,A -85,B 0,C 180,E1 25625.856,E2 25625.856} C_VEL
LIN {X 0,Y 559.885,Z 987.526,A -85,B 0,C 180,E1 25623.701,E2 25623.701} C_VEL
LIN {X 0,Y 559.902,Z 987.892,A -85,B 0,C 180,E1 25621.405,E2 25621.405} C_VEL
LIN {X 0,Y 559.918,Z 986.847,A -85,B 0,C 180,E1 25619.167,E2 25619.167} C_VEL
LIN {X 0,Y 559.916,Z 984.011,A -85,B 0,C 180,E1 25616.753,E2 25616.753} C_VEL
LIN {X 0,Y 559.937,Z 979.661,A -85,B 0,C 180,E1 25614.398,E2 25614.398} C_VEL
LIN {X 0,Y 559.954,Z 973.711,A -85,B 0,C 180,E1 25612.1,E2 25612.1} C_VEL
LIN {X 0,Y 560.037,Z 966.317,A -85,B 0,C 180,E1 25609.83,E2 25609.83} C_VEL
LIN {X 0,Y 560.175,Z 957.464,A -85,B 0,C 180,E1 25607.643,E2 25607.643} C_VEL
LIN {X 0,Y 560.399,Z 946.72,A -85,B 0,C 180,E1 25605.39,E2 25605.39} C_VEL
LIN {X 0,Y 560.683,Z 934.465,A -85,B 0,C 180,E1 25603.219,E2 25603.219} C_VEL
LIN {X 0,Y 561.095,Z 919.768,A -85,B 0,C 180,E1 25600.978,E2 25600.978} C_VEL
LIN {X 0,Y 561.597,Z 904.162,A -85,B 0,C 180,E1 25598.917,E2 25598.917} C_VEL
LIN {X 0,Y 562.182,Z 887.416,A -85,B 0,C 180,E1 25597.005,E2 25597.005} C_VEL
LIN {X 0,Y 562.847,Z 869.283,A -85,B 0,C 180,E1 25595.197,E2 25595.197} C_VEL
LIN {X 0,Y 563.567,Z 850.31,A -85,B 0,C 180,E1 25593.543,E2 25593.543} C_VEL
LIN {X 0,Y 564.346,Z 830.341,A -85,B 0,C 180,E1 25592.048,E2 25592.048} C_VEL
LIN {X 0,Y 565.143,Z 808.214,A -85,B 0,C 180,E1 25590.633,E2 25590.633} C_VEL
LIN {X 0,Y 565.877,Z 787.79,A -85,B 0,C 180,E1 25589.536,E2 25589.536} C_VEL
LIN {X 0,Y 566.517,Z 765.495,A -85,B 0,C 180,E1 25588.546,E2 25588.546} C_VEL
LIN {X 0,Y 567.181,Z 742.848,A -85,B 0,C 180,E1 25587.744,E2 25587.744} C_VEL
LIN {X 0,Y 567.613,Z 719.977,A -85,B 0,C 180,E1 25587.138,E2 25587.138} C_VEL
LIN {X 0,Y 567.971,Z 694.84,A -85,B 0,C 180,E1 25586.686,E2 25586.686} C_VEL
LIN {X 0,Y 569.447,Z 481.943,A -85,B 0,C 180,E1 25583.506,E2 25583.506} C_VEL
LIN {X 0,Y 570.097,Z 377.411,A -85,B 0,C 180,E1 25581.892,E2 25581.892} C_VEL
LIN {X 0,Y 564.975,Z 369.66,A -85,B 0,C 180,E1 25581.327,E2 25581.327} C_VEL
LIN {X 0,Y 562.845,Z 366.233,A -85,B 0,C 180,E1 25581.084,E2 25581.084} C_VEL
LIN {X 0,Y 560.731,Z 363.171,A -85,B 0,C 180,E1 25580.846,E2 25580.846} C_VEL
LIN {X 0,Y 560.337,Z 361.796,A -85,B 0,C 180,E1 25580.745,E2 25580.745} C_VEL
LIN {X 0,Y 560.269,Z 361.246,A -85,B 0,C 180,E1 25580.457,E2 25580.457} C_VEL
LIN {X 0,Y 560.252,Z 361.253,A -85,B 0,C 180,E1 25577.126,E2 25577.126} C_VEL
LIN {X 0,Y 560.273,Z 361.252,A -85,B 0,C 180,E1 25573.836,E2 25573.836} C_VEL
LIN {X 0,Y 560.266,Z 361.26,A -85,B 0,C 180,E1 25570.474,E2 25570.474} C_VEL
LIN {X 0,Y 560.273,Z 361.252,A -85,B 0,C 180,E1 25567.074,E2 25567.074} C_VEL
LIN {X 0,Y 560.267,Z 361.258,A -85,B 0,C 180,E1 25563.786,E2 25563.786} C_VEL
LIN {X 0,Y 560.27,Z 361.258,A -85,B 0,C 180,E1 25560.512,E2 25560.512} C_VEL
LIN {X 0,Y 560.262,Z 361.252,A -85,B 0,C 180,E1 25557.239,E2 25557.239} C_VEL
LIN {X 0,Y 560.269,Z 361.26,A -85,B 0,C 180,E1 25553.854,E2 25553.854} C_VEL
LIN {X 0,Y 560.279,Z 361.254,A -85,B 0,C 180,E1 25550.551,E2 25550.551} C_VEL
LIN {X 0,Y 560.244,Z 361.258,A -85,B 0,C 180,E1 25547.32,E2 25547.32} C_VEL
LIN {X 0,Y 560.28,Z 361.259,A -85,B 0,C 180,E1 25544.049,E2 25544.049} C_VEL
LIN {X 0,Y 560.241,Z 361.257,A -85,B 0,C 180,E1 25540.83,E2 25540.83} C_VEL
LIN {X 0,Y 560.241,Z 361.259,A -85,B 0,C 180,E1 25537.437,E2 25537.437} C_VEL
LIN {X 0,Y 560.263,Z 361.257,A -85,B 0,C 180,E1 25534.3,E2 25534.3} C_VEL
LIN {X 0,Y 560.218,Z 361.257,A -85,B 0,C 180,E1 25531.075,E2 25531.075} C_VEL
LIN {X 0,Y 560.274,Z 361.257,A -85,B 0,C 180,E1 25527.962,E2 25527.962} C_VEL
LIN {X 0,Y 560.203,Z 361.263,A -85,B 0,C 180,E1 25524.796,E2 25524.796} C_VEL
LIN {X 0,Y 560.267,Z 361.259,A -85,B 0,C 180,E1 25521.579,E2 25521.579} C_VEL
LIN {X 0,Y 560.195,Z 361.266,A -85,B 0,C 180,E1 25518.535,E2 25518.535} C_VEL
LIN {X 0,Y 560.244,Z 361.251,A -85,B 0,C 180,E1 25515.262,E2 25515.262} C_VEL
LIN {X 0,Y 560.31,Z 361.485,A -85,B 0,C 180,E1 25513.507,E2 25513.507} C_VEL
LIN {X 0,Y 561.459,Z 364.601,A -85,B 0,C 180,E1 25513.103,E2 25513.103} C_VEL
LIN {X 0,Y 568.011,Z 378.682,A -85,B 0,C 180,E1 25511.421,E2 25511.421} C_VEL
LIN {X 0,Y 568.238,Z 381.051,A -85,B 0,C 180,E1 25511.223,E2 25511.223} C_VEL
LIN {X 0,Y 568.117,Z 391.55,A -85,B 0,C 180,E1 25510.493,E2 25510.493} C_VEL
LIN {X 0,Y 570.263,Z 402.721,A -85,B 0,C 180,E1 25510.124,E2 25510.124} C_VEL
LIN {X 0,Y 568.752,Z 609.183,A -85,B 0,C 180,E1 25506.984,E2 25506.984} C_VEL
LIN {X 0,Y 567.809,Z 739.976,A -85,B 0,C 180,E1 25505.018,E2 25505.018} C_VEL
LIN {X 0,Y 567.32,Z 763.813,A -85,B 0,C 180,E1 25504.471,E2 25504.471} C_VEL
LIN {X 0,Y 566.848,Z 785.826,A -85,B 0,C 180,E1 25503.777,E2 25503.777} C_VEL
LIN {X 0,Y 566.167,Z 807.642,A -85,B 0,C 180,E1 25502.894,E2 25502.894} C_VEL
LIN {X 0,Y 565.507,Z 828.748,A -85,B 0,C 180,E1 25501.857,E2 25501.857} C_VEL
LIN {X 0,Y 564.725,Z 849.814,A -85,B 0,C 180,E1 25500.607,E2 25500.607} C_VEL
LIN {X 0,Y 563.96,Z 870.377,A -85,B 0,C 180,E1 25499.182,E2 25499.182} C_VEL
LIN {X 0,Y 563.25,Z 888.563,A -85,B 0,C 180,E1 25497.718,E2 25497.718} C_VEL
LIN {X 0,Y 562.525,Z 907.958,A -85,B 0,C 180,E1 25495.923,E2 25495.923} C_VEL
LIN {X 0,Y 561.904,Z 925.172,A -85,B 0,C 180,E1 25494.1,E2 25494.1} C_VEL
LIN {X 0,Y 561.36,Z 941.096,A -85,B 0,C 180,E1 25492.153,E2 25492.153} C_VEL
LIN {X 0,Y 560.903,Z 956.32,A -85,B 0,C 180,E1 25490.017,E2 25490.017} C_VEL
LIN {X 0,Y 560.561,Z 968.992,A -85,B 0,C 180,E1 25487.976,E2 25487.976} C_VEL
LIN {X 0,Y 560.297,Z 980.306,A -85,B 0,C 180,E1 25485.847,E2 25485.847} C_VEL
LIN {X 0,Y 560.126,Z 989.984,A -85,B 0,C 180,E1 25483.737,E2 25483.737} C_VEL
LIN {X 0,Y 560.022,Z 998.331,A -85,B 0,C 180,E1 25481.538,E2 25481.538} C_VEL
LIN {X 0,Y 559.945,Z 1004.861,A -85,B 0,C 180,E1 25479.458,E2 25479.458} C_VEL
LIN {X 0,Y 559.898,Z 1010.628,A -85,B 0,C 180,E1 25477.081,E2 25477.081} C_VEL
LIN {X 0,Y 559.911,Z 1014.272,A -85,B 0,C 180,E1 25475.023,E2 25475.023} C_VEL
LIN {X 0,Y 559.914,Z 1016.986,A -85,B 0,C 180,E1 25472.562,E2 25472.562} C_VEL
LIN {X 0,Y 559.887,Z 1017.916,A -85,B 0,C 180,E1 25470.412,E2 25470.412} C_VEL
LIN {X 0,Y 559.913,Z 1017.326,A -85,B 0,C 180,E1 25467.956,E2 25467.956} C_VEL
LIN {X 0,Y 559.909,Z 1015.28,A -85,B 0,C 180,E1 25465.702,E2 25465.702} C_VEL
LIN {X 0,Y 559.914,Z 1011.467,A -85,B 0,C 180,E1 25463.338,E2 25463.338} C_VEL
LIN {X 0,Y 559.946,Z 1006.814,A -85,B 0,C 180,E1 25461.273,E2 25461.273} C_VEL
LIN {X 0,Y 559.988,Z 999.777,A -85,B 0,C 180,E1 25458.885,E2 25458.885} C_VEL
LIN {X 0,Y 560.098,Z 992.124,A -85,B 0,C 180,E1 25456.795,E2 25456.795} C_VEL
LIN {X 0,Y 560.276,Z 981.902,A -85,B 0,C 180,E1 25454.477,E2 25454.477} C_VEL
LIN {X 0,Y 560.529,Z 970.841,A -85,B 0,C 180,E1 25452.352,E2 25452.352} C_VEL
LIN {X 0,Y 560.856,Z 957.78,A -85,B 0,C 180,E1 25450.205,E2 25450.205} C_VEL
LIN {X 0,Y 561.289,Z 943.348,A -85,B 0,C 180,E1 25448.138,E2 25448.138} C_VEL
LIN {X 0,Y 561.804,Z 927.979,A -85,B 0,C 180,E1 25446.232,E2 25446.232} C_VEL
LIN {X 0,Y 562.436,Z 910.161,A -85,B 0,C 180,E1 25444.298,E2 25444.298} C_VEL
LIN {X 0,Y 563.119,Z 892.257,A -85,B 0,C 180,E1 25442.596,E2 25442.596} C_VEL
LIN {X 0,Y 563.841,Z 873.4,A -85,B 0,C 180,E1 25441.051,E2 25441.051} C_VEL
LIN {X 0,Y 564.606,Z 852.68,A -85,B 0,C 180,E1 25439.576,E2 25439.576} C_VEL
LIN {X 0,Y 565.35,Z 832.918,A -85,B 0,C 180,E1 25438.379,E2 25438.379} C_VEL
LIN {X 0,Y 566.073,Z 810.171,A -85,B 0,C 180,E1 25437.22,E2 25437.22} C_VEL
LIN {X 0,Y 566.757,Z 788.897,A -85,B 0,C 180,E1 25436.336,E2 25436.336} C_VEL
LIN {X 0,Y 567.282,Z 766.029,A -85,B 0,C 180,E1 25435.591,E2 25435.591} C_VEL
LIN {X 0,Y 567.766,Z 743.551,A -85,B 0,C 180,E1 25435.046,E2 25435.046} C_VEL
LIN {X 0,Y 568.123,Z 701.783,A -85,B 0,C 180,E1 25434.391,E2 25434.391} C_VEL
LIN {X 0,Y 569.581,Z 492.547,A -85,B 0,C 180,E1 25431.255,E2 25431.255} C_VEL
LIN {X 0,Y 570.119,Z 401.01,A -85,B 0,C 180,E1 25429.836,E2 25429.836} C_VEL
LIN {X 0,Y 568.013,Z 390.671,A -85,B 0,C 180,E1 25429.466,E2 25429.466} C_VEL
LIN {X 0,Y 568.217,Z 379.137,A -85,B 0,C 180,E1 25428.632,E2 25428.632} C_VEL
LIN {X 0,Y 562.882,Z 367.733,A -85,B 0,C 180,E1 25427.276,E2 25427.276} C_VEL
LIN {X 0,Y 560.325,Z 361.562,A -85,B 0,C 180,E1 25426.515,E2 25426.515} C_VEL
LIN {X 0,Y 560.207,Z 361.252,A -85,B 0,C 180,E1 25425.321,E2 25425.321} C_VEL
LIN {X 0,Y 560.252,Z 361.259,A -85,B 0,C 180,E1 25422.069,E2 25422.069} C_VEL
LIN {X 0,Y 560.206,Z 361.253,A -85,B 0,C 180,E1 25419.052,E2 25419.052} C_VEL
LIN {X 0,Y 560.239,Z 361.248,A -85,B 0,C 180,E1 25415.829,E2 25415.829} C_VEL
LIN {X 0,Y 560.203,Z 361.263,A -85,B 0,C 180,E1 25412.801,E2 25412.801} C_VEL
LIN {X 0,Y 560.215,Z 361.26,A -85,B 0,C 180,E1 25409.439,E2 25409.439} C_VEL
LIN {X 0,Y 560.198,Z 361.262,A -85,B 0,C 180,E1 25406.606,E2 25406.606} C_VEL
LIN {X 0,Y 560.208,Z 361.261,A -85,B 0,C 180,E1 25403.208,E2 25403.208} C_VEL
LIN {X 0,Y 560.205,Z 361.261,A -85,B 0,C 180,E1 25400.367,E2 25400.367} C_VEL
LIN {X 0,Y 560.207,Z 361.261,A -85,B 0,C 180,E1 25396.913,E2 25396.913} C_VEL
LIN {X 0,Y 560.228,Z 361.259,A -85,B 0,C 180,E1 25393.942,E2 25393.942} C_VEL
LIN {X 0,Y 560.209,Z 361.26,A -85,B 0,C 180,E1 25390.697,E2 25390.697} C_VEL
LIN {X 0,Y 560.241,Z 361.259,A -85,B 0,C 180,E1 25387.692,E2 25387.692} C_VEL
LIN {X 0,Y 560.21,Z 361.26,A -85,B 0,C 180,E1 25384.401,E2 25384.401} C_VEL
LIN {X 0,Y 560.277,Z 361.259,A -85,B 0,C 180,E1 25381.227,E2 25381.227} C_VEL
LIN {X 0,Y 560.211,Z 361.259,A -85,B 0,C 180,E1 25378.056,E2 25378.056} C_VEL
LIN {X 0,Y 560.28,Z 361.258,A -85,B 0,C 180,E1 25374.88,E2 25374.88} C_VEL
LIN {X 0,Y 560.219,Z 361.256,A -85,B 0,C 180,E1 25371.687,E2 25371.687} C_VEL
LIN {X 0,Y 560.251,Z 361.256,A -85,B 0,C 180,E1 25368.365,E2 25368.365} C_VEL
LIN {X 0,Y 560.234,Z 361.259,A -85,B 0,C 180,E1 25365.29,E2 25365.29} C_VEL
LIN {X 0,Y 560.233,Z 361.254,A -85,B 0,C 180,E1 25361.908,E2 25361.908} C_VEL
LIN {X 0,Y 560.28,Z 361.257,A -85,B 0,C 180,E1 25358.663,E2 25358.663} C_VEL
LIN {X 0,Y 560.28,Z 361.254,A -85,B 0,C 180,E1 25356.227,E2 25356.227} C_VEL
LIN {X 0,Y 559.243,Z 361.381,A -85,B 0,C 180,E1 25355.44,E2 25355.44} C_VEL
LIN {X 0,Y 552.813,Z 362.184,A -85,B 0,C 180,E1 25353.228,E2 25353.228} C_VEL
LIN {X 0,Y 552.327,Z 362.25,A -85,B 0,C 180,E1 25352.652,E2 25352.652} C_VEL
LIN {X 0,Y 552.295,Z 362.246,A -85,B 0,C 180,E1 25349.298,E2 25349.298} C_VEL
LIN {X 0,Y 552.344,Z 362.242,A -85,B 0,C 180,E1 25345.988,E2 25345.988} C_VEL
LIN {X 0,Y 552.302,Z 362.248,A -85,B 0,C 180,E1 25342.794,E2 25342.794} C_VEL
LIN {X 0,Y 552.326,Z 362.241,A -85,B 0,C 180,E1 25339.466,E2 25339.466} C_VEL
LIN {X 0,Y 552.341,Z 362.246,A -85,B 0,C 180,E1 25336.086,E2 25336.086} C_VEL
LIN {X 0,Y 552.302,Z 362.243,A -85,B 0,C 180,E1 25332.75,E2 25332.75} C_VEL
LIN {X 0,Y 552.343,Z 362.243,A -85,B 0,C 180,E1 25329.443,E2 25329.443} C_VEL
LIN {X 0,Y 552.329,Z 362.25,A -85,B 0,C 180,E1 25326.033,E2 25326.033} C_VEL
LIN {X 0,Y 552.313,Z 362.241,A -85,B 0,C 180,E1 25322.643,E2 25322.643} C_VEL
LIN {X 0,Y 552.337,Z 362.235,A -85,B 0,C 180,E1 25319.373,E2 25319.373} C_VEL
LIN {X 0,Y 552.315,Z 362.248,A -85,B 0,C 180,E1 25316.093,E2 25316.093} C_VEL
LIN {X 0,Y 552.338,Z 362.243,A -85,B 0,C 180,E1 25312.675,E2 25312.675} C_VEL
LIN {X 0,Y 552.337,Z 362.247,A -85,B 0,C 180,E1 25309.232,E2 25309.232} C_VEL
LIN {X 0,Y 552.316,Z 362.224,A -85,B 0,C 180,E1 25305.86,E2 25305.86} C_VEL
LIN {X 0,Y 552.349,Z 362.461,A -85,B 0,C 180,E1 25303.963,E2 25303.963} C_VEL
LIN {X 0,Y 552.706,Z 363.882,A -85,B 0,C 180,E1 25303.782,E2 25303.782} C_VEL
LIN {X 0,Y 554.67,Z 366.938,A -85,B 0,C 180,E1 25303.549,E2 25303.549} C_VEL
LIN {X 0,Y 555.947,Z 368.745,A -85,B 0,C 180,E1 25303.402,E2 25303.402} C_VEL
LIN {X 0,Y 564.067,Z 381.097,A -85,B 0,C 180,E1 25302.474,E2 25302.474} C_VEL
LIN {X 0,Y 562.275,Z 589.279,A -85,B 0,C 180,E1 25299.279,E2 25299.279} C_VEL
LIN {X 0,Y 561.249,Z 711.252,A -85,B 0,C 180,E1 25297.424,E2 25297.424} C_VEL
LIN {X 0,Y 560.679,Z 734.904,A -85,B 0,C 180,E1 25296.865,E2 25296.865} C_VEL
LIN {X 0,Y 560.069,Z 757.872,A -85,B 0,C 180,E1 25296.12,E2 25296.12} C_VEL
LIN {X 0,Y 559.281,Z 779.306,A -85,B 0,C 180,E1 25295.228,E2 25295.228} C_VEL
LIN {X 0,Y 558.435,Z 801.447,A -85,B 0,C 180,E1 25294.104,E2 25294.104} C_VEL
LIN {X 0,Y 557.531,Z 822.491,A -85,B 0,C 180,E1 25292.824,E2 25292.824} C_VEL
LIN {X 0,Y 556.581,Z 843.865,A -85,B 0,C 180,E1 25291.284,E2 25291.284} C_VEL
LIN {X 0,Y 555.711,Z 863.003,A -85,B 0,C 180,E1 25289.688,E2 25289.688} C_VEL
LIN {X 0,Y 554.899,Z 881.135,A -85,B 0,C 180,E1 25287.932,E2 25287.932} C_VEL
LIN {X 0,Y 554.136,Z 898.908,A -85,B 0,C 180,E1 25285.962,E2 25285.962} C_VEL
LIN {X 0,Y 553.489,Z 915.238,A -85,B 0,C 180,E1 25283.879,E2 25283.879} C_VEL
LIN {X 0,Y 552.996,Z 929.46,A -85,B 0,C 180,E1 25281.785,E2 25281.785} C_VEL
LIN {X 0,Y 552.602,Z 942.417,A -85,B 0,C 180,E1 25279.573,E2 25279.573} C_VEL
LIN {X 0,Y 552.324,Z 953.636,A -85,B 0,C 180,E1 25277.344,E2 25277.344} C_VEL
LIN {X 0,Y 552.134,Z 963.112,A -85,B 0,C 180,E1 25275.096,E2 25275.096} C_VEL
LIN {X 0,Y 552,Z 971.148,A -85,B 0,C 180,E1 25272.825,E2 25272.825} C_VEL
LIN {X 0,Y 551.925,Z 977.523,A -85,B 0,C 180,E1 25270.526,E2 25270.526} C_VEL
LIN {X 0,Y 551.921,Z 982.28,A -85,B 0,C 180,E1 25268.309,E2 25268.309} C_VEL
LIN {X 0,Y 551.907,Z 985.711,A -85,B 0,C 180,E1 25265.934,E2 25265.934} C_VEL
LIN {X 0,Y 551.884,Z 987.516,A -85,B 0,C 180,E1 25263.742,E2 25263.742} C_VEL
LIN {X 0,Y 551.906,Z 987.873,A -85,B 0,C 180,E1 25261.307,E2 25261.307} C_VEL
LIN {X 0,Y 551.913,Z 986.69,A -85,B 0,C 180,E1 25258.912,E2 25258.912} C_VEL
LIN {X 0,Y 551.904,Z 983.865,A -85,B 0,C 180,E1 25256.58,E2 25256.58} C_VEL
LIN {X 0,Y 551.942,Z 979.576,A -85,B 0,C 180,E1 25254.25,E2 25254.25} C_VEL
LIN {X 0,Y 551.97,Z 973.785,A -85,B 0,C 180,E1 25251.981,E2 25251.981} C_VEL
LIN {X 0,Y 552.063,Z 966.427,A -85,B 0,C 180,E1 25249.685,E2 25249.685} C_VEL
LIN {X 0,Y 552.225,Z 957.629,A -85,B 0,C 180,E1 25247.47,E2 25247.47} C_VEL
LIN {X 0,Y 552.484,Z 946.94,A -85,B 0,C 180,E1 25245.189,E2 25245.189} C_VEL
LIN {X 0,Y 552.836,Z 934.735,A -85,B 0,C 180,E1 25242.988,E2 25242.988} C_VEL
LIN {X 0,Y 553.326,Z 920.109,A -85,B 0,C 180,E1 25240.718,E2 25240.718} C_VEL
LIN {X 0,Y 553.906,Z 904.717,A -85,B 0,C 180,E1 25238.651,E2 25238.651} C_VEL
LIN {X 0,Y 554.6,Z 887.968,A -85,B 0,C 180,E1 25236.702,E2 25236.702} C_VEL
LIN {X 0,Y 555.435,Z 869.13,A -85,B 0,C 180,E1 25234.796,E2 25234.796} C_VEL
LIN {X 0,Y 556.283,Z 850.12,A -85,B 0,C 180,E1 25233.121,E2 25233.121} C_VEL
LIN {X 0,Y 557.209,Z 829.995,A -85,B 0,C 180,E1 25231.599,E2 25231.599} C_VEL
LIN {X 0,Y 558.125,Z 808.75,A -85,B 0,C 180,E1 25230.226,E2 25230.226} C_VEL
LIN {X 0,Y 558.962,Z 788.336,A -85,B 0,C 180,E1 25229.114,E2 25229.114} C_VEL
LIN {X 0,Y 559.737,Z 765.898,A -85,B 0,C 180,E1 25228.103,E2 25228.103} C_VEL
LIN {X 0,Y 560.505,Z 743.276,A -85,B 0,C 180,E1 25227.292,E2 25227.292} C_VEL
LIN {X 0,Y 561.023,Z 720.057,A -85,B 0,C 180,E1 25226.67,E2 25226.67} C_VEL
LIN {X 0,Y 561.44,Z 694.755,A -85,B 0,C 180,E1 25226.212,E2 25226.212} C_VEL
LIN {X 0,Y 563.181,Z 481.76,A -85,B 0,C 180,E1 25222.995,E2 25222.995} C_VEL
LIN {X 0,Y 563.957,Z 380.84,A -85,B 0,C 180,E1 25221.422,E2 25221.422} C_VEL
LIN {X 0,Y 557.494,Z 371.258,A -85,B 0,C 180,E1 25220.691,E2 25220.691} C_VEL
LIN {X 0,Y 554.849,Z 367.113,A -85,B 0,C 180,E1 25220.38,E2 25220.38} C_VEL
LIN {X 0,Y 552.776,Z 364.006,A -85,B 0,C 180,E1 25220.136,E2 25220.136} C_VEL
LIN {X 0,Y 552.406,Z 362.663,A -85,B 0,C 180,E1 25220.005,E2 25220.005} C_VEL
LIN {X 0,Y 552.331,Z 362.198,A -85,B 0,C 180,E1 25219.567,E2 25219.567} C_VEL
LIN {X 0,Y 552.34,Z 362.249,A -85,B 0,C 180,E1 25216.188,E2 25216.188} C_VEL
LIN {X 0,Y 552.318,Z 362.247,A -85,B 0,C 180,E1 25212.866,E2 25212.866} C_VEL
LIN {X 0,Y 552.334,Z 362.244,A -85,B 0,C 180,E1 25209.587,E2 25209.587} C_VEL
LIN {X 0,Y 552.338,Z 362.25,A -85,B 0,C 180,E1 25206.236,E2 25206.236} C_VEL
LIN {X 0,Y 552.331,Z 362.243,A -85,B 0,C 180,E1 25202.802,E2 25202.802} C_VEL
LIN {X 0,Y 552.321,Z 362.246,A -85,B 0,C 180,E1 25199.482,E2 25199.482} C_VEL
LIN {X 0,Y 552.338,Z 362.247,A -85,B 0,C 180,E1 25196.16,E2 25196.16} C_VEL
LIN {X 0,Y 552.343,Z 362.242,A -85,B 0,C 180,E1 25192.721,E2 25192.721} C_VEL
LIN {X 0,Y 552.308,Z 362.246,A -85,B 0,C 180,E1 25189.359,E2 25189.359} C_VEL
LIN {X 0,Y 552.344,Z 362.248,A -85,B 0,C 180,E1 25185.998,E2 25185.998} C_VEL
LIN {X 0,Y 552.323,Z 362.244,A -85,B 0,C 180,E1 25182.621,E2 25182.621} C_VEL
LIN {X 0,Y 552.298,Z 362.247,A -85,B 0,C 180,E1 25179.328,E2 25179.328} C_VEL
LIN {X 0,Y 552.346,Z 362.243,A -85,B 0,C 180,E1 25176.079,E2 25176.079} C_VEL
LIN {X 0,Y 552.282,Z 362.248,A -85,B 0,C 180,E1 25172.857,E2 25172.857} C_VEL
LIN {X 0,Y 552.314,Z 362.251,A -85,B 0,C 180,E1 25169.544,E2 25169.544} C_VEL
LIN {X 0,Y 552.278,Z 362.251,A -85,B 0,C 180,E1 25166.484,E2 25166.484} C_VEL
LIN {X 0,Y 552.272,Z 362.253,A -85,B 0,C 180,E1 25163.054,E2 25163.054} C_VEL
LIN {X 0,Y 552.297,Z 362.254,A -85,B 0,C 180,E1 25159.979,E2 25159.979} C_VEL
LIN {X 0,Y 552.261,Z 362.256,A -85,B 0,C 180,E1 25156.673,E2 25156.673} C_VEL
LIN {X 0,Y 552.309,Z 362.502,A -85,B 0,C 180,E1 25154.202,E2 25154.202} C_VEL
LIN {X 0,Y 553.713,Z 365.863,A -85,B 0,C 180,E1 25153.756,E2 25153.756} C_VEL
LIN {X 0,Y 561.707,Z 383.072,A -85,B 0,C 180,E1 25151.655,E2 25151.655} C_VEL
LIN {X 0,Y 561.643,Z 391.655,A -85,B 0,C 180,E1 25151.057,E2 25151.057} C_VEL
LIN {X 0,Y 564.129,Z 404.348,A -85,B 0,C 180,E1 25150.625,E2 25150.625} C_VEL
LIN {X 0,Y 562.346,Z 610.837,A -85,B 0,C 180,E1 25147.451,E2 25147.451} C_VEL
LIN {X 0,Y 561.247,Z 740.169,A -85,B 0,C 180,E1 25145.486,E2 25145.486} C_VEL
LIN {X 0,Y 560.692,Z 763.811,A -85,B 0,C 180,E1 25144.937,E2 25144.937} C_VEL
LIN {X 0,Y 560.12,Z 785.841,A -85,B 0,C 180,E1 25144.238,E2 25144.238} C_VEL
LIN {X 0,Y 559.346,Z 807.639,A -85,B 0,C 180,E1 25143.347,E2 25143.347} C_VEL
LIN {X 0,Y 558.545,Z 828.748,A -85,B 0,C 180,E1 25142.302,E2 25142.302} C_VEL
LIN {X 0,Y 557.683,Z 849.016,A -85,B 0,C 180,E1 25141.09,E2 25141.09} C_VEL
LIN {X 0,Y 556.796,Z 868.905,A -85,B 0,C 180,E1 25139.713,E2 25139.713} C_VEL
LIN {X 0,Y 555.952,Z 887.506,A -85,B 0,C 180,E1 25138.208,E2 25138.208} C_VEL
LIN {X 0,Y 555.08,Z 906.771,A -85,B 0,C 180,E1 25136.42,E2 25136.42} C_VEL
LIN {X 0,Y 554.357,Z 923.641,A -85,B 0,C 180,E1 25134.625,E2 25134.625} C_VEL
LIN {X 0,Y 553.689,Z 939.977,A -85,B 0,C 180,E1 25132.624,E2 25132.624} C_VEL
LIN {X 0,Y 553.141,Z 954.904,A -85,B 0,C 180,E1 25130.531,E2 25130.531} C_VEL
LIN {X 0,Y 552.724,Z 967.72,A -85,B 0,C 180,E1 25128.458,E2 25128.458} C_VEL
LIN {X 0,Y 552.398,Z 979.786,A -85,B 0,C 180,E1 25126.188,E2 25126.188} C_VEL
LIN {X 0,Y 552.192,Z 989.524,A -85,B 0,C 180,E1 25124.045,E2 25124.045} C_VEL
LIN {X 0,Y 552.053,Z 998.332,A -85,B 0,C 180,E1 25121.706,E2 25121.706} C_VEL
LIN {X 0,Y 551.953,Z 1005.163,A -85,B 0,C 180,E1 25119.491,E2 25119.491} C_VEL
LIN {X 0,Y 551.902,Z 1010.628,A -85,B 0,C 180,E1 25117.184,E2 25117.184} C_VEL
LIN {X 0,Y 551.913,Z 1014.272,A -85,B 0,C 180,E1 25115.096,E2 25115.096} C_VEL
LIN {X 0,Y 551.911,Z 1016.986,A -85,B 0,C 180,E1 25112.599,E2 25112.599} C_VEL
LIN {X 0,Y 551.884,Z 1017.894,A -85,B 0,C 180,E1 25110.522,E2 25110.522} C_VEL
LIN {X 0,Y 551.912,Z 1017.393,A -85,B 0,C 180,E1 25108.031,E2 25108.031} C_VEL
LIN {X 0,Y 551.914,Z 1015.507,A -85,B 0,C 180,E1 25105.848,E2 25105.848} C_VEL
LIN {X 0,Y 551.917,Z 1011.674,A -85,B 0,C 180,E1 25103.345,E2 25103.345} C_VEL
LIN {X 0,Y 551.952,Z 1007.07,A -85,B 0,C 180,E1 25101.251,E2 25101.251} C_VEL
LIN {X 0,Y 552.007,Z 1000.131,A -85,B 0,C 180,E1 25098.828,E2 25098.828} C_VEL
LIN {X 0,Y 552.13,Z 992.534,A -85,B 0,C 180,E1 25096.708,E2 25096.708} C_VEL
LIN {X 0,Y 552.341,Z 982.419,A -85,B 0,C 180,E1 25094.356,E2 25094.356} C_VEL
LIN {X 0,Y 552.619,Z 972.004,A -85,B 0,C 180,E1 25092.308,E2 25092.308} C_VEL
LIN {X 0,Y 553.032,Z 958.491,A -85,B 0,C 180,E1 25090.023,E2 25090.023} C_VEL
LIN {X 0,Y 553.548,Z 944.073,A -85,B 0,C 180,E1 25087.912,E2 25087.912} C_VEL
LIN {X 0,Y 554.168,Z 928.241,A -85,B 0,C 180,E1 25085.915,E2 25085.915} C_VEL
LIN {X 0,Y 554.941,Z 910.161,A -85,B 0,C 180,E1 25083.925,E2 25083.925} C_VEL
LIN {X 0,Y 555.761,Z 891.951,A -85,B 0,C 180,E1 25082.174,E2 25082.174} C_VEL
LIN {X 0,Y 556.617,Z 872.907,A -85,B 0,C 180,E1 25080.599,E2 25080.599} C_VEL
LIN {X 0,Y 557.556,Z 851.793,A -85,B 0,C 180,E1 25079.089,E2 25079.089} C_VEL
LIN {X 0,Y 558.371,Z 832.914,A -85,B 0,C 180,E1 25077.937,E2 25077.937} C_VEL
LIN {X 0,Y 559.243,Z 809.991,A -85,B 0,C 180,E1 25076.759,E2 25076.759} C_VEL
LIN {X 0,Y 560.022,Z 788.894,A -85,B 0,C 180,E1 25075.876,E2 25075.876} C_VEL
LIN {X 0,Y 560.635,Z 765.947,A -85,B 0,C 180,E1 25075.122,E2 25075.122} C_VEL
LIN {X 0,Y 561.211,Z 743.209,A -85,B 0,C 180,E1 25074.569,E2 25074.569} C_VEL
LIN {X 0,Y 561.657,Z 697.086,A -85,B 0,C 180,E1 25073.845,E2 25073.845} C_VEL
LIN {X 0,Y 563.364,Z 489.061,A -85,B 0,C 180,E1 25070.689,E2 25070.689} C_VEL
LIN {X 0,Y 563.983,Z 402.782,A -85,B 0,C 180,E1 25069.337,E2 25069.337} C_VEL
LIN {X 0,Y 561.523,Z 390.881,A -85,B 0,C 180,E1 25068.911,E2 25068.911} C_VEL
LIN {X 0,Y 561.609,Z 382.833,A -85,B 0,C 180,E1 25068.318,E2 25068.318} C_VEL
LIN {X 0,Y 553.716,Z 365.856,A -85,B 0,C 180,E1 25066.243,E2 25066.243} C_VEL
LIN {X 0,Y 552.302,Z 362.428,A -85,B 0,C 180,E1 25065.775,E2 25065.775} C_VEL
LIN {X 0,Y 552.283,Z 362.235,A -85,B 0,C 180,E1 25062.899,E2 25062.899} C_VEL
LIN {X 0,Y 552.269,Z 362.238,A -85,B 0,C 180,E1 25059.541,E2 25059.541} C_VEL
LIN {X 0,Y 552.308,Z 362.244,A -85,B 0,C 180,E1 25056.426,E2 25056.426} C_VEL
LIN {X 0,Y 552.261,Z 362.253,A -85,B 0,C 180,E1 25053.243,E2 25053.243} C_VEL
LIN {X 0,Y 552.325,Z 362.233,A -85,B 0,C 180,E1 25050.092,E2 25050.092} C_VEL
LIN {X 0,Y 552.254,Z 362.251,A -85,B 0,C 180,E1 25046.912,E2 25046.912} C_VEL
LIN {X 0,Y 552.32,Z 362.247,A -85,B 0,C 180,E1 25043.664,E2 25043.664} C_VEL
LIN {X 0,Y 552.258,Z 362.25,A -85,B 0,C 180,E1 25040.562,E2 25040.562} C_VEL
LIN {X 0,Y 552.298,Z 362.25,A -85,B 0,C 180,E1 25037.271,E2 25037.271} C_VEL
LIN {X 0,Y 552.267,Z 362.248,A -85,B 0,C 180,E1 25034.254,E2 25034.254} C_VEL
LIN {X 0,Y 552.279,Z 362.249,A -85,B 0,C 180,E1 25030.852,E2 25030.852} C_VEL
LIN {X 0,Y 552.291,Z 362.247,A -85,B 0,C 180,E1 25027.803,E2 25027.803} C_VEL
LIN {X 0,Y 552.273,Z 362.249,A -85,B 0,C 180,E1 25024.465,E2 25024.465} C_VEL
LIN {X 0,Y 552.337,Z 362.247,A -85,B 0,C 180,E1 25021.244,E2 25021.244} C_VEL
LIN {X 0,Y 552.273,Z 362.248,A -85,B 0,C 180,E1 25018.028,E2 25018.028} C_VEL
LIN {X 0,Y 552.336,Z 362.247,A -85,B 0,C 180,E1 25014.807,E2 25014.807} C_VEL
LIN {X 0,Y 552.281,Z 362.245,A -85,B 0,C 180,E1 25011.672,E2 25011.672} C_VEL
LIN {X 0,Y 552.306,Z 362.245,A -85,B 0,C 180,E1 25008.301,E2 25008.301} C_VEL
LIN {X 0,Y 552.307,Z 362.249,A -85,B 0,C 180,E1 25005.155,E2 25005.155} C_VEL
LIN {X 0,Y 552.292,Z 362.243,A -85,B 0,C 180,E1 25001.857,E2 25001.857} C_VEL
LIN {X 0,Y 552.341,Z 362.246,A -85,B 0,C 180,E1 24998.662,E2 24998.662} C_VEL
LIN {X 0,Y 552.288,Z 362.246,A -85,B 0,C 180,E1 24995.393,E2 24995.393} C_VEL
LIN {X 0,Y 552.327,Z 362.25,A -85,B 0,C 180,E1 24992.652,E2 24992.652} C_VEL
LIN {X 0,Y 551.38,Z 362.376,A -85,B 0,C 180,E1 24991.853,E2 24991.853} C_VEL
LIN {X 0,Y 544.885,Z 363.17,A -85,B 0,C 180,E1 24989.609,E2 24989.609} C_VEL
LIN {X 0,Y 544.357,Z 363.237,A -85,B 0,C 180,E1 24989.024,E2 24989.024} C_VEL
LIN {X 0,Y 544.382,Z 363.231,A -85,B 0,C 180,E1 24985.676,E2 24985.676} C_VEL
LIN {X 0,Y 544.396,Z 363.236,A -85,B 0,C 180,E1 24982.326,E2 24982.326} C_VEL
LIN {X 0,Y 544.363,Z 363.233,A -85,B 0,C 180,E1 24979.01,E2 24979.01} C_VEL
LIN {X 0,Y 544.403,Z 363.233,A -85,B 0,C 180,E1 24975.74,E2 24975.74} C_VEL
LIN {X 0,Y 544.372,Z 363.233,A -85,B 0,C 180,E1 24972.407,E2 24972.407} C_VEL
LIN {X 0,Y 544.374,Z 363.234,A -85,B 0,C 180,E1 24968.908,E2 24968.908} C_VEL
LIN {X 0,Y 544.4,Z 363.231,A -85,B 0,C 180,E1 24965.548,E2 24965.548} C_VEL
LIN {X 0,Y 544.376,Z 363.233,A -85,B 0,C 180,E1 24962.179,E2 24962.179} C_VEL
LIN {X 0,Y 544.389,Z 363.224,A -85,B 0,C 180,E1 24958.759,E2 24958.759} C_VEL
LIN {X 0,Y 544.398,Z 363.223,A -85,B 0,C 180,E1 24955.361,E2 24955.361} C_VEL
LIN {X 0,Y 544.377,Z 363.233,A -85,B 0,C 180,E1 24952.001,E2 24952.001} C_VEL
LIN {X 0,Y 544.4,Z 363.229,A -85,B 0,C 180,E1 24948.611,E2 24948.611} C_VEL
LIN {X 0,Y 544.399,Z 363.222,A -85,B 0,C 180,E1 24945.223,E2 24945.223} C_VEL
LIN {X 0,Y 544.451,Z 363.581,A -85,B 0,C 180,E1 24944.677,E2 24944.677} C_VEL
LIN {X 0,Y 544.953,Z 365.312,A -85,B 0,C 180,E1 24944.491,E2 24944.491} C_VEL
LIN {X 0,Y 546.997,Z 368.198,A -85,B 0,C 180,E1 24944.245,E2 24944.245} C_VEL
LIN {X 0,Y 557.948,Z 384.486,A -85,B 0,C 180,E1 24942.957,E2 24942.957} C_VEL
LIN {X 0,Y 555.88,Z 592.765,A -85,B 0,C 180,E1 24939.727,E2 24939.727} C_VEL
LIN {X 0,Y 554.726,Z 711.232,A -85,B 0,C 180,E1 24937.906,E2 24937.906} C_VEL
LIN {X 0,Y 554.093,Z 734.732,A -85,B 0,C 180,E1 24937.348,E2 24937.348} C_VEL
LIN {X 0,Y 553.388,Z 757.374,A -85,B 0,C 180,E1 24936.611,E2 24936.611} C_VEL
LIN {X 0,Y 552.508,Z 778.931,A -85,B 0,C 180,E1 24935.709,E2 24935.709} C_VEL
LIN {X 0,Y 551.503,Z 801.194,A -85,B 0,C 180,E1 24934.572,E2 24934.572} C_VEL
LIN {X 0,Y 550.487,Z 822.299,A -85,B 0,C 180,E1 24933.277,E2 24933.277} C_VEL
LIN {X 0,Y 549.367,Z 843.744,A -85,B 0,C 180,E1 24931.718,E2 24931.718} C_VEL
LIN {X 0,Y 548.372,Z 862.893,A -85,B 0,C 180,E1 24930.101,E2 24930.101} C_VEL
LIN {X 0,Y 547.423,Z 881.054,A -85,B 0,C 180,E1 24928.322,E2 24928.322} C_VEL
LIN {X 0,Y 546.527,Z 898.845,A -85,B 0,C 180,E1 24926.326,E2 24926.326} C_VEL
LIN {X 0,Y 545.761,Z 915.565,A -85,B 0,C 180,E1 24924.159,E2 24924.159} C_VEL
LIN {X 0,Y 545.178,Z 930.074,A -85,B 0,C 180,E1 24921.985,E2 24921.985} C_VEL
LIN {X 0,Y 544.708,Z 943.146,A -85,B 0,C 180,E1 24919.699,E2 24919.699} C_VEL
LIN {X 0,Y 544.378,Z 954.569,A -85,B 0,C 180,E1 24917.372,E2 24917.372} C_VEL
LIN {X 0,Y 544.162,Z 963.875,A -85,B 0,C 180,E1 24915.091,E2 24915.091} C_VEL
LIN {X 0,Y 544.012,Z 972.066,A -85,B 0,C 180,E1 24912.675,E2 24912.675} C_VEL
LIN {X 0,Y 543.928,Z 978.008,A -85,B 0,C 180,E1 24910.452,E2 24910.452} C_VEL
LIN {X 0,Y 543.909,Z 982.832,A -85,B 0,C 180,E1 24908.086,E2 24908.086} C_VEL
LIN {X 0,Y 543.915,Z 986.046,A -85,B 0,C 180,E1 24905.681,E2 24905.681} C_VEL
LIN {X 0,Y 543.91,Z 987.744,A -85,B 0,C 180,E1 24903.23,E2 24903.23} C_VEL
LIN {X 0,Y 543.914,Z 987.804,A -85,B 0,C 180,E1 24900.965,E2 24900.965} C_VEL
LIN {X 0,Y 543.905,Z 986.232,A -85,B 0,C 180,E1 24898.402,E2 24898.402} C_VEL
LIN {X 0,Y 543.896,Z 983.124,A -85,B 0,C 180,E1 24896.006,E2 24896.006} C_VEL
LIN {X 0,Y 543.926,Z 978.287,A -85,B 0,C 180,E1 24893.574,E2 24893.574} C_VEL
LIN {X 0,Y 544.019,Z 972.329,A -85,B 0,C 180,E1 24891.324,E2 24891.324} C_VEL
LIN {X 0,Y 544.164,Z 964.05,A -85,B 0,C 180,E1 24888.866,E2 24888.866} C_VEL
LIN {X 0,Y 544.368,Z 954.879,A -85,B 0,C 180,E1 24886.61,E2 24886.61} C_VEL
LIN {X 0,Y 544.694,Z 943.516,A -85,B 0,C 180,E1 24884.281,E2 24884.281} C_VEL
LIN {X 0,Y 545.145,Z 930.685,A -85,B 0,C 180,E1 24882.025,E2 24882.025} C_VEL
LIN {X 0,Y 545.728,Z 916.291,A -85,B 0,C 180,E1 24879.852,E2 24879.852} C_VEL
LIN {X 0,Y 546.459,Z 900.39,A -85,B 0,C 180,E1 24877.772,E2 24877.772} C_VEL
LIN {X 0,Y 547.306,Z 883.503,A -85,B 0,C 180,E1 24875.84,E2 24875.84} C_VEL
LIN {X 0,Y 548.214,Z 865.479,A -85,B 0,C 180,E1 24874.051,E2 24874.051} C_VEL
LIN {X 0,Y 549.264,Z 845.81,A -85,B 0,C 180,E1 24872.357,E2 24872.357} C_VEL
LIN {X 0,Y 550.325,Z 825.074,A -85,B 0,C 180,E1 24870.821,E2 24870.821} C_VEL
LIN {X 0,Y 551.396,Z 803.923,A -85,B 0,C 180,E1 24869.493,E2 24869.493} C_VEL
LIN {X 0,Y 552.397,Z 781.31,A -85,B 0,C 180,E1 24868.31,E2 24868.31} C_VEL
LIN {X 0,Y 553.268,Z 760.244,A -85,B 0,C 180,E1 24867.412,E2 24867.412} C_VEL
LIN {X 0,Y 554.037,Z 736.405,A -85,B 0,C 180,E1 24866.609,E2 24866.609} C_VEL
LIN {X 0,Y 554.663,Z 713.365,A -85,B 0,C 180,E1 24866.048,E2 24866.048} C_VEL
LIN {X 0,Y 555.142,Z 672.797,A -85,B 0,C 180,E1 24865.397,E2 24865.397} C_VEL
LIN {X 0,Y 557.144,Z 462.992,A -85,B 0,C 180,E1 24862.183,E2 24862.183} C_VEL
LIN {X 0,Y 557.827,Z 384.29,A -85,B 0,C 180,E1 24860.939,E2 24860.939} C_VEL
LIN {X 0,Y 549.459,Z 371.999,A -85,B 0,C 180,E1 24859.964,E2 24859.964} C_VEL
LIN {X 0,Y 547.113,Z 368.259,A -85,B 0,C 180,E1 24859.678,E2 24859.678} C_VEL
LIN {X 0,Y 544.926,Z 365.255,A -85,B 0,C 180,E1 24859.416,E2 24859.416} C_VEL
LIN {X 0,Y 544.443,Z 363.648,A -85,B 0,C 180,E1 24859.248,E2 24859.248} C_VEL
LIN {X 0,Y 544.365,Z 363.183,A -85,B 0,C 180,E1 24858.861,E2 24858.861} C_VEL
LIN {X 0,Y 544.401,Z 363.228,A -85,B 0,C 180,E1 24855.445,E2 24855.445} C_VEL
LIN {X 0,Y 544.398,Z 363.234,A -85,B 0,C 180,E1 24851.979,E2 24851.979} C_VEL
LIN {X 0,Y 544.384,Z 363.236,A -85,B 0,C 180,E1 24848.663,E2 24848.663} C_VEL
LIN {X 0,Y 544.399,Z 363.228,A -85,B 0,C 180,E1 24845.269,E2 24845.269} C_VEL
LIN {X 0,Y 544.389,Z 363.238,A -85,B 0,C 180,E1 24841.79,E2 24841.79} C_VEL
LIN {X 0,Y 544.394,Z 363.235,A -85,B 0,C 180,E1 24838.527,E2 24838.527} C_VEL
LIN {X 0,Y 544.385,Z 363.232,A -85,B 0,C 180,E1 24835.154,E2 24835.154} C_VEL
LIN {X 0,Y 544.38,Z 363.238,A -85,B 0,C 180,E1 24831.657,E2 24831.657} C_VEL
LIN {X 0,Y 544.402,Z 363.234,A -85,B 0,C 180,E1 24828.345,E2 24828.345} C_VEL
LIN {X 0,Y 544.366,Z 363.235,A -85,B 0,C 180,E1 24825.048,E2 24825.048} C_VEL
LIN {X 0,Y 544.384,Z 363.239,A -85,B 0,C 180,E1 24821.696,E2 24821.696} C_VEL
LIN {X 0,Y 544.385,Z 363.232,A -85,B 0,C 180,E1 24818.449,E2 24818.449} C_VEL
LIN {X 0,Y 544.348,Z 363.239,A -85,B 0,C 180,E1 24815.126,E2 24815.126} C_VEL
LIN {X 0,Y 544.405,Z 363.238,A -85,B 0,C 180,E1 24811.835,E2 24811.835} C_VEL
LIN {X 0,Y 544.338,Z 363.238,A -85,B 0,C 180,E1 24808.666,E2 24808.666} C_VEL
LIN {X 0,Y 544.349,Z 363.242,A -85,B 0,C 180,E1 24805.292,E2 24805.292} C_VEL
LIN {X 0,Y 544.348,Z 363.242,A -85,B 0,C 180,E1 24802.158,E2 24802.158} C_VEL
LIN {X 0,Y 544.323,Z 363.245,A -85,B 0,C 180,E1 24798.864,E2 24798.864} C_VEL
LIN {X 0,Y 544.393,Z 363.223,A -85,B 0,C 180,E1 24795.593,E2 24795.593} C_VEL
LIN {X 0,Y 544.375,Z 363.522,A -85,B 0,C 180,E1 24794.886,E2 24794.886} C_VEL
LIN {X 0,Y 545.944,Z 367.173,A -85,B 0,C 180,E1 24794.398,E2 24794.398} C_VEL
LIN {X 0,Y 555.177,Z 386.849,A -85,B 0,C 180,E1 24791.964,E2 24791.964} C_VEL
LIN {X 0,Y 555.203,Z 391.687,A -85,B 0,C 180,E1 24791.638,E2 24791.638} C_VEL
LIN {X 0,Y 558.035,Z 406.248,A -85,B 0,C 180,E1 24791.132,E2 24791.132} C_VEL
LIN {X 0,Y 555.977,Z 612.618,A -85,B 0,C 180,E1 24787.927,E2 24787.927} C_VEL
LIN {X 0,Y 554.725,Z 740.167,A -85,B 0,C 180,E1 24785.967,E2 24785.967} C_VEL
LIN {X 0,Y 554.109,Z 763.679,A -85,B 0,C 180,E1 24785.418,E2 24785.418} C_VEL
LIN {X 0,Y 553.434,Z 785.466,A -85,B 0,C 180,E1 24784.725,E2 24784.725} C_VEL
LIN {X 0,Y 552.6,Z 806.764,A -85,B 0,C 180,E1 24783.851,E2 24783.851} C_VEL
LIN {X 0,Y 551.718,Z 826.522,A -85,B 0,C 180,E1 24782.875,E2 24782.875} C_VEL
LIN {X 0,Y 550.688,Z 848.027,A -85,B 0,C 180,E1 24781.597,E2 24781.597} C_VEL
LIN {X 0,Y 549.67,Z 868.16,A -85,B 0,C 180,E1 24780.198,E2 24780.198} C_VEL
LIN {X 0,Y 548.623,Z 887.867,A -85,B 0,C 180,E1 24778.587,E2 24778.587} C_VEL
LIN {X 0,Y 547.596,Z 907.197,A -85,B 0,C 180,E1 24776.765,E2 24776.765} C_VEL
LIN {X 0,Y 546.747,Z 924.652,A -85,B 0,C 180,E1 24774.876,E2 24774.876} C_VEL
LIN {X 0,Y 545.97,Z 940.824,A -85,B 0,C 180,E1 24772.848,E2 24772.848} C_VEL
LIN {X 0,Y 545.304,Z 956.324,A -85,B 0,C 180,E1 24770.615,E2 24770.615} C_VEL
LIN {X 0,Y 544.835,Z 968.988,A -85,B 0,C 180,E1 24768.513,E2 24768.513} C_VEL
LIN {X 0,Y 544.477,Z 980.309,A -85,B 0,C 180,E1 24766.32,E2 24766.32} C_VEL
LIN {X 0,Y 544.228,Z 990.441,A -85,B 0,C 180,E1 24764.038,E2 24764.038} C_VEL
LIN {X 0,Y 544.074,Z 998.689,A -85,B 0,C 180,E1 24761.773,E2 24761.773} C_VEL
LIN {X 0,Y 543.965,Z 1005.767,A -85,B 0,C 180,E1 24759.418,E2 24759.418} C_VEL
LIN {X 0,Y 543.905,Z 1010.835,A -85,B 0,C 180,E1 24757.184,E2 24757.184} C_VEL
LIN {X 0,Y 543.912,Z 1014.431,A -85,B 0,C 180,E1 24755.065,E2 24755.065} C_VEL
LIN {X 0,Y 543.913,Z 1017.054,A -85,B 0,C 180,E1 24752.532,E2 24752.532} C_VEL
LIN {X 0,Y 543.892,Z 1017.939,A -85,B 0,C 180,E1 24750.319,E2 24750.319} C_VEL
LIN {X 0,Y 543.914,Z 1017.326,A -85,B 0,C 180,E1 24747.896,E2 24747.896} C_VEL
LIN {X 0,Y 543.909,Z 1015.393,A -85,B 0,C 180,E1 24745.681,E2 24745.681} C_VEL
LIN {X 0,Y 543.914,Z 1011.674,A -85,B 0,C 180,E1 24743.247,E2 24743.247} C_VEL
LIN {X 0,Y 543.964,Z 1007.07,A -85,B 0,C 180,E1 24741.122,E2 24741.122} C_VEL
LIN {X 0,Y 544.033,Z 1000.131,A -85,B 0,C 180,E1 24738.663,E2 24738.663} C_VEL
LIN {X 0,Y 544.17,Z 992.535,A -85,B 0,C 180,E1 24736.509,E2 24736.509} C_VEL
LIN {X 0,Y 544.418,Z 982.418,A -85,B 0,C 180,E1 24734.123,E2 24734.123} C_VEL
LIN {X 0,Y 544.745,Z 972.006,A -85,B 0,C 180,E1 24732.044,E2 24732.044} C_VEL
LIN {X 0,Y 545.235,Z 958.492,A -85,B 0,C 180,E1 24729.725,E2 24729.725} C_VEL
LIN {X 0,Y 545.837,Z 944.249,A -85,B 0,C 180,E1 24727.608,E2 24727.608} C_VEL
LIN {X 0,Y 546.544,Z 928.445,A -85,B 0,C 180,E1 24725.583,E2 24725.583} C_VEL
LIN {X 0,Y 547.462,Z 910.162,A -85,B 0,C 180,E1 24723.541,E2 24723.541} C_VEL
LIN {X 0,Y 548.427,Z 891.952,A -85,B 0,C 180,E1 24721.769,E2 24721.769} C_VEL
LIN {X 0,Y 549.409,Z 872.661,A -85,B 0,C 180,E1 24720.155,E2 24720.155} C_VEL
LIN {X 0,Y 550.535,Z 851.113,A -85,B 0,C 180,E1 24718.604,E2 24718.604} C_VEL
LIN {X 0,Y 551.471,Z 831.906,A -85,B 0,C 180,E1 24717.425,E2 24717.425} C_VEL
LIN {X 0,Y 552.433,Z 810.348,A -85,B 0,C 180,E1 24716.312,E2 24716.312} C_VEL
LIN {X 0,Y 553.252,Z 790.503,A -85,B 0,C 180,E1 24715.468,E2 24715.468} C_VEL
LIN {X 0,Y 554.003,Z 767.055,A -85,B 0,C 180,E1 24714.677,E2 24714.677} C_VEL
LIN {X 0,Y 554.607,Z 745.335,A -85,B 0,C 180,E1 24714.134,E2 24714.134} C_VEL
LIN {X 0,Y 555.056,Z 712.354,A -85,B 0,C 180,E1 24713.586,E2 24713.586} C_VEL
LIN {X 0,Y 557.058,Z 501.783,A -85,B 0,C 180,E1 24710.365,E2 24710.365} C_VEL
LIN {X 0,Y 557.889,Z 404.571,A -85,B 0,C 180,E1 24708.827,E2 24708.827} C_VEL
LIN {X 0,Y 555.076,Z 390.771,A -85,B 0,C 180,E1 24708.321,E2 24708.321} C_VEL
LIN {X 0,Y 555.035,Z 386.483,A -85,B 0,C 180,E1 24707.995,E2 24707.995} C_VEL
LIN {X 0,Y 547.077,Z 369.768,A -85,B 0,C 180,E1 24705.911,E2 24705.911} C_VEL
LIN {X 0,Y 544.394,Z 363.614,A -85,B 0,C 180,E1 24705.113,E2 24705.113} C_VEL
LIN {X 0,Y 544.386,Z 363.2,A -85,B 0,C 180,E1 24704.556,E2 24704.556} C_VEL
LIN {X 0,Y 544.327,Z 363.244,A -85,B 0,C 180,E1 24701.306,E2 24701.306} C_VEL
LIN {X 0,Y 544.38,Z 363.237,A -85,B 0,C 180,E1 24698.015,E2 24698.015} C_VEL
LIN {X 0,Y 544.328,Z 363.225,A -85,B 0,C 180,E1 24694.816,E2 24694.816} C_VEL
LIN {X 0,Y 544.326,Z 363.23,A -85,B 0,C 180,E1 24691.321,E2 24691.321} C_VEL
LIN {X 0,Y 544.352,Z 363.237,A -85,B 0,C 180,E1 24688.287,E2 24688.287} C_VEL
LIN {X 0,Y 544.318,Z 363.241,A -85,B 0,C 180,E1 24684.991,E2 24684.991} C_VEL
LIN {X 0,Y 544.397,Z 363.239,A -85,B 0,C 180,E1 24681.777,E2 24681.777} C_VEL
LIN {X 0,Y 544.32,Z 363.24,A -85,B 0,C 180,E1 24678.528,E2 24678.528} C_VEL
LIN {X 0,Y 544.362,Z 363.235,A -85,B 0,C 180,E1 24675.227,E2 24675.227} C_VEL
LIN {X 0,Y 544.331,Z 363.239,A -85,B 0,C 180,E1 24672.195,E2 24672.195} C_VEL
LIN {X 0,Y 544.341,Z 363.235,A -85,B 0,C 180,E1 24668.769,E2 24668.769} C_VEL
LIN {X 0,Y 544.349,Z 363.239,A -85,B 0,C 180,E1 24665.798,E2 24665.798} C_VEL
LIN {X 0,Y 544.336,Z 363.234,A -85,B 0,C 180,E1 24662.421,E2 24662.421} C_VEL
LIN {X 0,Y 544.392,Z 363.236,A -85,B 0,C 180,E1 24659.263,E2 24659.263} C_VEL
LIN {X 0,Y 544.336,Z 363.237,A -85,B 0,C 180,E1 24655.997,E2 24655.997} C_VEL
LIN {X 0,Y 544.396,Z 363.231,A -85,B 0,C 180,E1 24652.719,E2 24652.719} C_VEL
LIN {X 0,Y 544.348,Z 363.238,A -85,B 0,C 180,E1 24649.522,E2 24649.522} C_VEL
LIN {X 0,Y 544.355,Z 363.234,A -85,B 0,C 180,E1 24646.077,E2 24646.077} C_VEL
LIN {X 0,Y 544.388,Z 363.24,A -85,B 0,C 180,E1 24642.91,E2 24642.91} C_VEL
LIN {X 0,Y 544.349,Z 363.236,A -85,B 0,C 180,E1 24639.574,E2 24639.574} C_VEL
LIN {X 0,Y 544.405,Z 363.232,A -85,B 0,C 180,E1 24636.283,E2 24636.283} C_VEL
LIN {X 0,Y 544.363,Z 363.238,A -85,B 0,C 180,E1 24632.965,E2 24632.965} C_VEL
LIN {X 0,Y 544.36,Z 363.235,A -85,B 0,C 180,E1 24629.469,E2 24629.469} C_VEL
LIN {X 0,Y 544.357,Z 363.237,A -85,B 0,C 180,E1 24629.024,E2 24629.024} C_VEL
LIN {X 0,Y 543.391,Z 363.361,A -85,B 0,C 180,E1 24628.214,E2 24628.214} C_VEL
LIN {X 0,Y 536.873,Z 364.17,A -85,B 0,C 180,E1 24625.877,E2 24625.877} C_VEL
LIN {X 0,Y 536.422,Z 364.221,A -85,B 0,C 180,E1 24625.343,E2 24625.343} C_VEL
LIN {X 0,Y 536.467,Z 364.221,A -85,B 0,C 180,E1 24622.026,E2 24622.026} C_VEL
LIN {X 0,Y 536.426,Z 364.223,A -85,B 0,C 180,E1 24618.684,E2 24618.684} C_VEL
LIN {X 0,Y 536.44,Z 364.221,A -85,B 0,C 180,E1 24615.207,E2 24615.207} C_VEL
LIN {X 0,Y 536.465,Z 364.225,A -85,B 0,C 180,E1 24611.796,E2 24611.796} C_VEL
LIN {X 0,Y 536.429,Z 364.226,A -85,B 0,C 180,E1 24608.478,E2 24608.478} C_VEL
LIN {X 0,Y 536.454,Z 364.215,A -85,B 0,C 180,E1 24605.028,E2 24605.028} C_VEL
LIN {X 0,Y 536.462,Z 364.226,A -85,B 0,C 180,E1 24601.577,E2 24601.577} C_VEL
LIN {X 0,Y 536.433,Z 364.216,A -85,B 0,C 180,E1 24598.252,E2 24598.252} C_VEL
LIN {X 0,Y 536.459,Z 364.208,A -85,B 0,C 180,E1 24594.813,E2 24594.813} C_VEL
LIN {X 0,Y 536.463,Z 364.21,A -85,B 0,C 180,E1 24591.422,E2 24591.422} C_VEL
LIN {X 0,Y 536.436,Z 364.2,A -85,B 0,C 180,E1 24588.019,E2 24588.019} C_VEL
LIN {X 0,Y 536.483,Z 364.418,A -85,B 0,C 180,E1 24585.483,E2 24585.483} C_VEL
LIN {X 0,Y 536.869,Z 365.922,A -85,B 0,C 180,E1 24585.285,E2 24585.285} C_VEL
LIN {X 0,Y 538.853,Z 368.999,A -85,B 0,C 180,E1 24585.025,E2 24585.025} C_VEL
LIN {X 0,Y 540.04,Z 370.478,A -85,B 0,C 180,E1 24584.88,E2 24584.88} C_VEL
LIN {X 0,Y 542.849,Z 374.496,A -85,B 0,C 180,E1 24584.533,E2 24584.533} C_VEL
LIN {X 0,Y 551.865,Z 388.167,A -85,B 0,C 180,E1 24583.446,E2 24583.446} C_VEL
LIN {X 0,Y 549.512,Z 596.835,A -85,B 0,C 180,E1 24580.177,E2 24580.177} C_VEL
LIN {X 0,Y 548.237,Z 711.365,A -85,B 0,C 180,E1 24578.396,E2 24578.396} C_VEL
LIN {X 0,Y 547.556,Z 734.436,A -85,B 0,C 180,E1 24577.845,E2 24577.845} C_VEL
LIN {X 0,Y 546.724,Z 757.561,A -85,B 0,C 180,E1 24577.087,E2 24577.087} C_VEL
LIN {X 0,Y 545.773,Z 778.553,A -85,B 0,C 180,E1 24576.202,E2 24576.202} C_VEL
LIN {X 0,Y 544.615,Z 800.935,A -85,B 0,C 180,E1 24575.052,E2 24575.052} C_VEL
LIN {X 0,Y 543.476,Z 822.107,A -85,B 0,C 180,E1 24573.741,E2 24573.741} C_VEL
LIN {X 0,Y 542.184,Z 843.623,A -85,B 0,C 180,E1 24572.163,E2 24572.163} C_VEL
LIN {X 0,Y 541.03,Z 863.368,A -85,B 0,C 180,E1 24570.473,E2 24570.473} C_VEL
LIN {X 0,Y 539.935,Z 881.486,A -85,B 0,C 180,E1 24568.67,E2 24568.67} C_VEL
LIN {X 0,Y 538.939,Z 898.782,A -85,B 0,C 180,E1 24566.7,E2 24566.7} C_VEL
LIN {X 0,Y 538.096,Z 915.099,A -85,B 0,C 180,E1 24564.559,E2 24564.559} C_VEL
LIN {X 0,Y 537.398,Z 930.007,A -85,B 0,C 180,E1 24562.299,E2 24562.299} C_VEL
LIN {X 0,Y 536.859,Z 942.861,A -85,B 0,C 180,E1 24560.023,E2 24560.023} C_VEL
LIN {X 0,Y 536.462,Z 954.502,A -85,B 0,C 180,E1 24557.621,E2 24557.621} C_VEL
LIN {X 0,Y 536.204,Z 963.812,A -85,B 0,C 180,E1 24555.307,E2 24555.307} C_VEL
LIN {X 0,Y 536.026,Z 972.007,A -85,B 0,C 180,E1 24552.857,E2 24552.857} C_VEL
LIN {X 0,Y 535.94,Z 977.958,A -85,B 0,C 180,E1 24550.602,E2 24550.602} C_VEL
LIN {X 0,Y 535.917,Z 982.786,A -85,B 0,C 180,E1 24548.203,E2 24548.203} C_VEL
LIN {X 0,Y 535.915,Z 986.02,A -85,B 0,C 180,E1 24545.764,E2 24545.764} C_VEL
LIN {X 0,Y 535.909,Z 987.739,A -85,B 0,C 180,E1 24543.277,E2 24543.277} C_VEL
LIN {X 0,Y 535.914,Z 987.811,A -85,B 0,C 180,E1 24540.98,E2 24540.98} C_VEL
LIN {X 0,Y 535.906,Z 986.264,A -85,B 0,C 180,E1 24538.378,E2 24538.378} C_VEL
LIN {X 0,Y 535.899,Z 983.155,A -85,B 0,C 180,E1 24535.935,E2 24535.935} C_VEL
LIN {X 0,Y 535.933,Z 978.353,A -85,B 0,C 180,E1 24533.475,E2 24533.475} C_VEL
LIN {X 0,Y 536.032,Z 972.398,A -85,B 0,C 180,E1 24531.188,E2 24531.188} C_VEL
LIN {X 0,Y 536.203,Z 964.134,A -85,B 0,C 180,E1 24528.69,E2 24528.69} C_VEL
LIN {X 0,Y 536.449,Z 954.965,A -85,B 0,C 180,E1 24526.397,E2 24526.397} C_VEL
LIN {X 0,Y 536.837,Z 943.475,A -85,B 0,C 180,E1 24524.005,E2 24524.005} C_VEL
LIN {X 0,Y 537.355,Z 930.779,A -85,B 0,C 180,E1 24521.74,E2 24521.74} C_VEL
LIN {X 0,Y 538.054,Z 915.872,A -85,B 0,C 180,E1 24519.46,E2 24519.46} C_VEL
LIN {X 0,Y 538.922,Z 899.151,A -85,B 0,C 180,E1 24517.255,E2 24517.255} C_VEL
LIN {X 0,Y 539.933,Z 881.557,A -85,B 0,C 180,E1 24515.247,E2 24515.247} C_VEL
LIN {X 0,Y 541.043,Z 863.147,A -85,B 0,C 180,E1 24513.416,E2 24513.416} C_VEL
LIN {X 0,Y 542.173,Z 843.885,A -85,B 0,C 180,E1 24511.768,E2 24511.768} C_VEL
LIN {X 0,Y 543.439,Z 822.658,A -85,B 0,C 180,E1 24510.207,E2 24510.207} C_VEL
LIN {X 0,Y 544.61,Z 801.075,A -85,B 0,C 180,E1 24508.866,E2 24508.866} C_VEL
LIN {X 0,Y 545.778,Z 778.432,A -85,B 0,C 180,E1 24507.702,E2 24507.702} C_VEL
LIN {X 0,Y 546.757,Z 756.483,A -85,B 0,C 180,E1 24506.783,E2 24506.783} C_VEL
LIN {X 0,Y 547.596,Z 733.367,A -85,B 0,C 180,E1 24506.035,E2 24506.035} C_VEL
LIN {X 0,Y 548.258,Z 710.268,A -85,B 0,C 180,E1 24505.493,E2 24505.493} C_VEL
LIN {X 0,Y 550.642,Z 494.281,A -85,B 0,C 180,E1 24502.14,E2 24502.14} C_VEL
LIN {X 0,Y 551.751,Z 387.783,A -85,B 0,C 180,E1 24500.447,E2 24500.447} C_VEL
LIN {X 0,Y 542.032,Z 373.571,A -85,B 0,C 180,E1 24499.281,E2 24499.281} C_VEL
LIN {X 0,Y 539.121,Z 369.225,A -85,B 0,C 180,E1 24498.914,E2 24498.914} C_VEL
LIN {X 0,Y 537.023,Z 366.347,A -85,B 0,C 180,E1 24498.65,E2 24498.65} C_VEL
LIN {X 0,Y 536.571,Z 364.931,A -85,B 0,C 180,E1 24498.525,E2 24498.525} C_VEL
LIN {X 0,Y 536.461,Z 364.203,A -85,B 0,C 180,E1 24498.248,E2 24498.248} C_VEL
LIN {X 0,Y 536.435,Z 364.211,A -85,B 0,C 180,E1 24494.905,E2 24494.905} C_VEL
LIN {X 0,Y 536.461,Z 364.221,A -85,B 0,C 180,E1 24491.504,E2 24491.504} C_VEL
LIN {X 0,Y 536.46,Z 364.223,A -85,B 0,C 180,E1 24488.036,E2 24488.036} C_VEL
LIN {X 0,Y 536.449,Z 364.221,A -85,B 0,C 180,E1 24484.597,E2 24484.597} C_VEL
LIN {X 0,Y 536.459,Z 364.221,A -85,B 0,C 180,E1 24481.175,E2 24481.175} C_VEL
LIN {X 0,Y 536.447,Z 364.221,A -85,B 0,C 180,E1 24477.757,E2 24477.757} C_VEL
LIN {X 0,Y 536.46,Z 364.221,A -85,B 0,C 180,E1 24474.331,E2 24474.331} C_VEL
LIN {X 0,Y 536.444,Z 364.222,A -85,B 0,C 180,E1 24470.993,E2 24470.993} C_VEL
LIN {X 0,Y 536.433,Z 364.227,A -85,B 0,C 180,E1 24467.514,E2 24467.514} C_VEL
LIN {X 0,Y 536.465,Z 364.224,A -85,B 0,C 180,E1 24464.21,E2 24464.21} C_VEL
LIN {X 0,Y 536.425,Z 364.225,A -85,B 0,C 180,E1 24460.85,E2 24460.85} C_VEL
LIN {X 0,Y 536.419,Z 364.226,A -85,B 0,C 180,E1 24457.32,E2 24457.32} C_VEL
LIN {X 0,Y 536.464,Z 364.223,A -85,B 0,C 180,E1 24454.025,E2 24454.025} C_VEL
LIN {X 0,Y 536.401,Z 364.223,A -85,B 0,C 180,E1 24450.767,E2 24450.767} C_VEL
LIN {X 0,Y 536.423,Z 364.231,A -85,B 0,C 180,E1 24447.407,E2 24447.407} C_VEL
LIN {X 0,Y 536.404,Z 364.231,A -85,B 0,C 180,E1 24444.308,E2 24444.308} C_VEL
LIN {X 0,Y 536.386,Z 364.233,A -85,B 0,C 180,E1 24440.946,E2 24440.946} C_VEL
LIN {X 0,Y 536.427,Z 364.227,A -85,B 0,C 180,E1 24437.855,E2 24437.855} C_VEL
LIN {X 0,Y 536.483,Z 364.444,A -85,B 0,C 180,E1 24435.621,E2 24435.621} C_VEL
LIN {X 0,Y 537.666,Z 367.612,A -85,B 0,C 180,E1 24435.187,E2 24435.187} C_VEL
LIN {X 0,Y 546.264,Z 385.527,A -85,B 0,C 180,E1 24432.916,E2 24432.916} C_VEL
LIN {X 0,Y 548.707,Z 391.136,A -85,B 0,C 180,E1 24432.254,E2 24432.254} C_VEL
LIN {X 0,Y 551.988,Z 408.028,A -85,B 0,C 180,E1 24431.652,E2 24431.652} C_VEL
LIN {X 0,Y 549.648,Z 614.272,A -85,B 0,C 180,E1 24428.416,E2 24428.416} C_VEL
LIN {X 0,Y 548.241,Z 740.352,A -85,B 0,C 180,E1 24426.457,E2 24426.457} C_VEL
LIN {X 0,Y 547.557,Z 763.808,A -85,B 0,C 180,E1 24425.903,E2 24425.903} C_VEL
LIN {X 0,Y 546.776,Z 785.793,A -85,B 0,C 180,E1 24425.198,E2 24425.198} C_VEL
LIN {X 0,Y 545.817,Z 807.482,A -85,B 0,C 180,E1 24424.294,E2 24424.294} C_VEL
LIN {X 0,Y 544.81,Z 827.644,A -85,B 0,C 180,E1 24423.283,E2 24423.283} C_VEL
LIN {X 0,Y 543.655,Z 848.474,A -85,B 0,C 180,E1 24422.023,E2 24422.023} C_VEL
LIN {X 0,Y 542.486,Z 868.899,A -85,B 0,C 180,E1 24420.579,E2 24420.579} C_VEL
LIN {X 0,Y 541.332,Z 887.907,A -85,B 0,C 180,E1 24419.005,E2 24419.005} C_VEL
LIN {X 0,Y 540.172,Z 907.161,A -85,B 0,C 180,E1 24417.167,E2 24417.167} C_VEL
LIN {X 0,Y 539.217,Z 924.269,A -85,B 0,C 180,E1 24415.292,E2 24415.292} C_VEL
LIN {X 0,Y 538.34,Z 939.977,A -85,B 0,C 180,E1 24413.306,E2 24413.306} C_VEL
LIN {X 0,Y 537.603,Z 954.908,A -85,B 0,C 180,E1 24411.153,E2 24411.153} C_VEL
LIN {X 0,Y 537.053,Z 967.716,A -85,B 0,C 180,E1 24409.017,E2 24409.017} C_VEL
LIN {X 0,Y 536.602,Z 979.789,A -85,B 0,C 180,E1 24406.678,E2 24406.678} C_VEL
LIN {X 0,Y 536.318,Z 989.522,A -85,B 0,C 180,E1 24404.469,E2 24404.469} C_VEL
LIN {X 0,Y 536.106,Z 998.334,A -85,B 0,C 180,E1 24402.06,E2 24402.06} C_VEL
LIN {X 0,Y 535.972,Z 1005.163,A -85,B 0,C 180,E1 24399.777,E2 24399.777} C_VEL
LIN {X 0,Y 535.916,Z 1010.629,A -85,B 0,C 180,E1 24397.399,E2 24397.399} C_VEL
LIN {X 0,Y 535.916,Z 1014.272,A -85,B 0,C 180,E1 24395.248,E2 24395.248} C_VEL
LIN {X 0,Y 535.905,Z 1016.986,A -85,B 0,C 180,E1 24392.677,E2 24392.677} C_VEL
LIN {X 0,Y 535.885,Z 1017.894,A -85,B 0,C 180,E1 24390.538,E2 24390.538} C_VEL
LIN {X 0,Y 535.913,Z 1017.393,A -85,B 0,C 180,E1 24387.972,E2 24387.972} C_VEL
LIN {X 0,Y 535.911,Z 1015.506,A -85,B 0,C 180,E1 24385.724,E2 24385.724} C_VEL
LIN {X 0,Y 535.911,Z 1011.674,A -85,B 0,C 180,E1 24383.146,E2 24383.146} C_VEL
LIN {X 0,Y 535.976,Z 1007.071,A -85,B 0,C 180,E1 24380.988,E2 24380.988} C_VEL
LIN {X 0,Y 536.065,Z 1000.13,A -85,B 0,C 180,E1 24378.492,E2 24378.492} C_VEL
LIN {X 0,Y 536.219,Z 992.446,A -85,B 0,C 180,E1 24376.281,E2 24376.281} C_VEL
LIN {X 0,Y 536.505,Z 982.417,A -85,B 0,C 180,E1 24373.882,E2 24373.882} C_VEL
LIN {X 0,Y 536.873,Z 971.996,A -85,B 0,C 180,E1 24371.769,E2 24371.769} C_VEL
LIN {X 0,Y 537.442,Z 958.49,A -85,B 0,C 180,E1 24369.418,E2 24369.418} C_VEL
LIN {X 0,Y 538.144,Z 944.249,A -85,B 0,C 180,E1 24367.27,E2 24367.27} C_VEL
LIN {X 0,Y 538.954,Z 928.446,A -85,B 0,C 180,E1 24365.216,E2 24365.216} C_VEL
LIN {X 0,Y 540.002,Z 910.162,A -85,B 0,C 180,E1 24363.146,E2 24363.146} C_VEL
LIN {X 0,Y 541.109,Z 892.1,A -85,B 0,C 180,E1 24361.366,E2 24361.366} C_VEL
LIN {X 0,Y 542.227,Z 872.658,A -85,B 0,C 180,E1 24359.718,E2 24359.718} C_VEL
LIN {X 0,Y 543.47,Z 851.969,A -85,B 0,C 180,E1 24358.208,E2 24358.208} C_VEL
LIN {X 0,Y 544.512,Z 832.909,A -85,B 0,C 180,E1 24357.018,E2 24357.018} C_VEL
LIN {X 0,Y 545.675,Z 810.352,A -85,B 0,C 180,E1 24355.838,E2 24355.838} C_VEL
LIN {X 0,Y 546.558,Z 791.109,A -85,B 0,C 180,E1 24355.01,E2 24355.01} C_VEL
LIN {X 0,Y 547.416,Z 767.751,A -85,B 0,C 180,E1 24354.208,E2 24354.208} C_VEL
LIN {X 0,Y 548.079,Z 746.309,A -85,B 0,C 180,E1 24353.663,E2 24353.663} C_VEL
LIN {X 0,Y 548.592,Z 714.926,A -85,B 0,C 180,E1 24353.128,E2 24353.128} C_VEL
LIN {X 0,Y 550.865,Z 504.474,A -85,B 0,C 180,E1 24349.874,E2 24349.874} C_VEL
LIN {X 0,Y 551.836,Z 406.349,A -85,B 0,C 180,E1 24348.305,E2 24348.305} C_VEL
LIN {X 0,Y 548.672,Z 390.703,A -85,B 0,C 180,E1 24347.719,E2 24347.719} C_VEL
LIN {X 0,Y 540.176,Z 372.546,A -85,B 0,C 180,E1 24345.449,E2 24345.449} C_VEL
LIN {X 0,Y 536.533,Z 364.67,A -85,B 0,C 180,E1 24344.396,E2 24344.396} C_VEL
LIN {X 0,Y 536.408,Z 364.187,A -85,B 0,C 180,E1 24343.9,E2 24343.9} C_VEL
LIN {X 0,Y 536.407,Z 364.223,A -85,B 0,C 180,E1 24340.826,E2 24340.826} C_VEL
LIN {X 0,Y 536.39,Z 364.232,A -85,B 0,C 180,E1 24337.421,E2 24337.421} C_VEL
LIN {X 0,Y 536.451,Z 364.213,A -85,B 0,C 180,E1 24334.126,E2 24334.126} C_VEL
LIN {X 0,Y 536.379,Z 364.217,A -85,B 0,C 180,E1 24330.963,E2 24330.963} C_VEL
LIN {X 0,Y 536.433,Z 364.229,A -85,B 0,C 180,E1 24327.716,E2 24327.716} C_VEL
LIN {X 0,Y 536.383,Z 364.231,A -85,B 0,C 180,E1 24324.553,E2 24324.553} C_VEL
LIN {X 0,Y 536.39,Z 364.227,A -85,B 0,C 180,E1 24321.085,E2 24321.085} C_VEL
LIN {X 0,Y 536.425,Z 364.228,A -85,B 0,C 180,E1 24317.911,E2 24317.911} C_VEL
LIN {X 0,Y 536.385,Z 364.225,A -85,B 0,C 180,E1 24314.68,E2 24314.68} C_VEL
LIN {X 0,Y 536.454,Z 364.223,A -85,B 0,C 180,E1 24311.503,E2 24311.503} C_VEL
LIN {X 0,Y 536.389,Z 364.224,A -85,B 0,C 180,E1 24308.224,E2 24308.224} C_VEL
LIN {X 0,Y 536.431,Z 364.226,A -85,B 0,C 180,E1 24304.918,E2 24304.918} C_VEL
LIN {X 0,Y 536.411,Z 364.224,A -85,B 0,C 180,E1 24301.709,E2 24301.709} C_VEL
LIN {X 0,Y 536.4,Z 364.225,A -85,B 0,C 180,E1 24298.291,E2 24298.291} C_VEL
LIN {X 0,Y 536.462,Z 364.224,A -85,B 0,C 180,E1 24294.974,E2 24294.974} C_VEL
LIN {X 0,Y 536.401,Z 364.222,A -85,B 0,C 180,E1 24291.747,E2 24291.747} C_VEL
LIN {X 0,Y 536.437,Z 364.222,A -85,B 0,C 180,E1 24288.387,E2 24288.387} C_VEL
LIN {X 0,Y 536.423,Z 364.226,A -85,B 0,C 180,E1 24285.205,E2 24285.205} C_VEL
LIN {X 0,Y 536.415,Z 364.22,A -85,B 0,C 180,E1 24281.863,E2 24281.863} C_VEL
LIN {X 0,Y 536.467,Z 364.221,A -85,B 0,C 180,E1 24278.573,E2 24278.573} C_VEL
LIN {X 0,Y 536.412,Z 364.224,A -85,B 0,C 180,E1 24275.321,E2 24275.321} C_VEL
LIN {X 0,Y 536.455,Z 364.217,A -85,B 0,C 180,E1 24271.986,E2 24271.986} C_VEL
LIN {X 0,Y 536.44,Z 364.227,A -85,B 0,C 180,E1 24268.666,E2 24268.666} C_VEL
LIN {X 0,Y 536.422,Z 364.221,A -85,B 0,C 180,E1 24265.343,E2 24265.343} C_VEL
LIN {X 0,Y 535.437,Z 364.35,A -85,B 0,C 180,E1 24264.52,E2 24264.52} C_VEL
LIN {X 0,Y 528.984,Z 365.155,A -85,B 0,C 180,E1 24262.149,E2 24262.149} C_VEL
LIN {X 0,Y 528.515,Z 365.209,A -85,B 0,C 180,E1 24261.607,E2 24261.607} C_VEL
LIN {X 0,Y 528.52,Z 365.212,A -85,B 0,C 180,E1 24258.184,E2 24258.184} C_VEL
LIN {X 0,Y 528.487,Z 365.212,A -85,B 0,C 180,E1 24254.807,E2 24254.807} C_VEL
LIN {X 0,Y 528.529,Z 365.209,A -85,B 0,C 180,E1 24251.455,E2 24251.455} C_VEL
LIN {X 0,Y 528.524,Z 365.212,A -85,B 0,C 180,E1 24247.934,E2 24247.934} C_VEL
LIN {X 0,Y 528.493,Z 365.207,A -85,B 0,C 180,E1 24244.575,E2 24244.575} C_VEL
LIN {X 0,Y 528.525,Z 365.21,A -85,B 0,C 180,E1 24241.216,E2 24241.216} C_VEL
LIN {X 0,Y 528.523,Z 365.208,A -85,B 0,C 180,E1 24237.703,E2 24237.703} C_VEL
LIN {X 0,Y 528.497,Z 365.203,A -85,B 0,C 180,E1 24234.231,E2 24234.231} C_VEL
LIN {X 0,Y 528.521,Z 365.197,A -85,B 0,C 180,E1 24230.829,E2 24230.829} C_VEL
LIN {X 0,Y 528.518,Z 365.17,A -85,B 0,C 180,E1 24227.388,E2 24227.388} C_VEL
LIN {X 0,Y 528.528,Z 365.321,A -85,B 0,C 180,E1 24226.312,E2 24226.312} C_VEL
LIN {X 0,Y 528.841,Z 366.698,A -85,B 0,C 180,E1 24226.104,E2 24226.104} C_VEL
LIN {X 0,Y 530.652,Z 369.718,A -85,B 0,C 180,E1 24225.851,E2 24225.851} C_VEL
LIN {X 0,Y 532.145,Z 371.433,A -85,B 0,C 180,E1 24225.664,E2 24225.664} C_VEL
LIN {X 0,Y 534.905,Z 375.445,A -85,B 0,C 180,E1 24225.307,E2 24225.307} C_VEL
LIN {X 0,Y 545.826,Z 391.742,A -85,B 0,C 180,E1 24223.947,E2 24223.947} C_VEL
LIN {X 0,Y 543.171,Z 601.665,A -85,B 0,C 180,E1 24220.625,E2 24220.625} C_VEL
LIN {X 0,Y 541.795,Z 711.337,A -85,B 0,C 180,E1 24218.901,E2 24218.901} C_VEL
LIN {X 0,Y 541.065,Z 734.132,A -85,B 0,C 180,E1 24218.354,E2 24218.354} C_VEL
LIN {X 0,Y 540.12,Z 757.04,A -85,B 0,C 180,E1 24217.602,E2 24217.602} C_VEL
LIN {X 0,Y 539.076,Z 778.166,A -85,B 0,C 180,E1 24216.707,E2 24216.707} C_VEL
LIN {X 0,Y 537.781,Z 800.661,A -85,B 0,C 180,E1 24215.545,E2 24215.545} C_VEL
LIN {X 0,Y 536.498,Z 821.915,A -85,B 0,C 180,E1 24214.218,E2 24214.218} C_VEL
LIN {X 0,Y 535.095,Z 842.834,A -85,B 0,C 180,E1 24212.674,E2 24212.674} C_VEL
LIN {X 0,Y 533.782,Z 862.674,A -85,B 0,C 180,E1 24210.963,E2 24210.963} C_VEL
LIN {X 0,Y 532.525,Z 880.905,A -85,B 0,C 180,E1 24209.136,E2 24209.136} C_VEL
LIN {X 0,Y 531.382,Z 898.713,A -85,B 0,C 180,E1 24207.085,E2 24207.085} C_VEL
LIN {X 0,Y 530.422,Z 915.033,A -85,B 0,C 180,E1 24204.914,E2 24204.914} C_VEL
LIN {X 0,Y 529.622,Z 929.943,A -85,B 0,C 180,E1 24202.621,E2 24202.621} C_VEL
LIN {X 0,Y 529.001,Z 942.803,A -85,B 0,C 180,E1 24200.313,E2 24200.313} C_VEL
LIN {X 0,Y 528.552,Z 954.434,A -85,B 0,C 180,E1 24197.876,E2 24197.876} C_VEL
LIN {X 0,Y 528.252,Z 963.749,A -85,B 0,C 180,E1 24195.529,E2 24195.529} C_VEL
LIN {X 0,Y 528.043,Z 972.112,A -85,B 0,C 180,E1 24192.986,E2 24192.986} C_VEL
LIN {X 0,Y 527.947,Z 978.175,A -85,B 0,C 180,E1 24190.642,E2 24190.642} C_VEL
LIN {X 0,Y 527.914,Z 983.058,A -85,B 0,C 180,E1 24188.134,E2 24188.134} C_VEL
LIN {X 0,Y 527.914,Z 986.238,A -85,B 0,C 180,E1 24185.611,E2 24185.611} C_VEL
LIN {X 0,Y 527.91,Z 987.784,A -85,B 0,C 180,E1 24183.083,E2 24183.083} C_VEL
LIN {X 0,Y 527.917,Z 987.767,A -85,B 0,C 180,E1 24180.746,E2 24180.746} C_VEL
LIN {X 0,Y 527.909,Z 986.166,A -85,B 0,C 180,E1 24178.226,E2 24178.226} C_VEL
LIN {X 0,Y 527.908,Z 983.046,A -85,B 0,C 180,E1 24175.767,E2 24175.767} C_VEL
LIN {X 0,Y 527.942,Z 978.419,A -85,B 0,C 180,E1 24173.373,E2 24173.373} C_VEL
LIN {X 0,Y 528.055,Z 972.118,A -85,B 0,C 180,E1 24170.926,E2 24170.926} C_VEL
LIN {X 0,Y 528.26,Z 963.766,A -85,B 0,C 180,E1 24168.386,E2 24168.386} C_VEL
LIN {X 0,Y 528.557,Z 954.421,A -85,B 0,C 180,E1 24166.031,E2 24166.031} C_VEL
LIN {X 0,Y 528.989,Z 942.915,A -85,B 0,C 180,E1 24163.618,E2 24163.618} C_VEL
LIN {X 0,Y 529.635,Z 929.484,A -85,B 0,C 180,E1 24161.213,E2 24161.213} C_VEL
LIN {X 0,Y 530.446,Z 914.686,A -85,B 0,C 180,E1 24158.946,E2 24158.946} C_VEL
LIN {X 0,Y 531.394,Z 898.663,A -85,B 0,C 180,E1 24156.819,E2 24156.819} C_VEL
LIN {X 0,Y 532.544,Z 880.576,A -85,B 0,C 180,E1 24154.738,E2 24154.738} C_VEL
LIN {X 0,Y 533.814,Z 862.166,A -85,B 0,C 180,E1 24152.901,E2 24152.901} C_VEL
LIN {X 0,Y 535.1,Z 842.8,A -85,B 0,C 180,E1 24151.234,E2 24151.234} C_VEL
LIN {X 0,Y 536.523,Z 821.479,A -85,B 0,C 180,E1 24149.662,E2 24149.662} C_VEL
LIN {X 0,Y 537.821,Z 800.079,A -85,B 0,C 180,E1 24148.332,E2 24148.332} C_VEL
LIN {X 0,Y 539.072,Z 778.265,A -85,B 0,C 180,E1 24147.207,E2 24147.207} C_VEL
LIN {X 0,Y 540.146,Z 756.303,A -85,B 0,C 180,E1 24146.28,E2 24146.28} C_VEL
LIN {X 0,Y 541.105,Z 733.15,A -85,B 0,C 180,E1 24145.528,E2 24145.528} C_VEL
LIN {X 0,Y 541.823,Z 710.152,A -85,B 0,C 180,E1 24144.986,E2 24144.986} C_VEL
LIN {X 0,Y 544.479,Z 495.739,A -85,B 0,C 180,E1 24141.622,E2 24141.622} C_VEL
LIN {X 0,Y 545.648,Z 391.36,A -85,B 0,C 180,E1 24139.94,E2 24139.94} C_VEL
LIN {X 0,Y 534.654,Z 375.165,A -85,B 0,C 180,E1 24138.57,E2 24138.57} C_VEL
LIN {X 0,Y 532.007,Z 371.135,A -85,B 0,C 180,E1 24138.222,E2 24138.222} C_VEL
LIN {X 0,Y 529.158,Z 367.453,A -85,B 0,C 180,E1 24137.853,E2 24137.853} C_VEL
LIN {X 0,Y 528.666,Z 365.992,A -85,B 0,C 180,E1 24137.728,E2 24137.728} C_VEL
LIN {X 0,Y 528.522,Z 365.236,A -85,B 0,C 180,E1 24137.506,E2 24137.506} C_VEL
LIN {X 0,Y 528.521,Z 365.196,A -85,B 0,C 180,E1 24134.014,E2 24134.014} C_VEL
LIN {X 0,Y 528.508,Z 365.216,A -85,B 0,C 180,E1 24130.575,E2 24130.575} C_VEL
LIN {X 0,Y 528.518,Z 365.208,A -85,B 0,C 180,E1 24127.064,E2 24127.064} C_VEL
LIN {X 0,Y 528.51,Z 365.213,A -85,B 0,C 180,E1 24123.688,E2 24123.688} C_VEL
LIN {X 0,Y 528.524,Z 365.21,A -85,B 0,C 180,E1 24120.217,E2 24120.217} C_VEL
LIN {X 0,Y 528.521,Z 365.206,A -85,B 0,C 180,E1 24116.747,E2 24116.747} C_VEL
LIN {X 0,Y 528.498,Z 365.214,A -85,B 0,C 180,E1 24113.343,E2 24113.343} C_VEL
LIN {X 0,Y 528.516,Z 365.216,A -85,B 0,C 180,E1 24109.867,E2 24109.867} C_VEL
LIN {X 0,Y 528.526,Z 365.212,A -85,B 0,C 180,E1 24106.433,E2 24106.433} C_VEL
LIN {X 0,Y 528.484,Z 365.213,A -85,B 0,C 180,E1 24103.061,E2 24103.061} C_VEL
LIN {X 0,Y 528.502,Z 365.211,A -85,B 0,C 180,E1 24099.629,E2 24099.629} C_VEL
LIN {X 0,Y 528.514,Z 365.209,A -85,B 0,C 180,E1 24096.301,E2 24096.301} C_VEL
LIN {X 0,Y 528.467,Z 365.216,A -85,B 0,C 180,E1 24092.995,E2 24092.995} C_VEL
LIN {X 0,Y 528.51,Z 365.217,A -85,B 0,C 180,E1 24089.661,E2 24089.661} C_VEL
LIN {X 0,Y 528.464,Z 365.219,A -85,B 0,C 180,E1 24086.464,E2 24086.464} C_VEL
LIN {X 0,Y 528.453,Z 365.221,A -85,B 0,C 180,E1 24082.984,E2 24082.984} C_VEL
LIN {X 0,Y 528.517,Z 365.212,A -85,B 0,C 180,E1 24079.679,E2 24079.679} C_VEL
LIN {X 0,Y 528.464,Z 365.358,A -85,B 0,C 180,E1 24076.441,E2 24076.441} C_VEL
LIN {X 0,Y 528.761,Z 366.623,A -85,B 0,C 180,E1 24076.205,E2 24076.205} C_VEL
LIN {X 0,Y 530.913,Z 370.997,A -85,B 0,C 180,E1 24075.603,E2 24075.603} C_VEL
LIN {X 0,Y 539.994,Z 389.98,A -85,B 0,C 180,E1 24073.153,E2 24073.153} C_VEL
LIN {X 0,Y 543.309,Z 395.794,A -85,B 0,C 180,E1 24072.686,E2 24072.686} C_VEL
LIN {X 0,Y 545.986,Z 409.902,A -85,B 0,C 180,E1 24072.182,E2 24072.182} C_VEL
LIN {X 0,Y 543.357,Z 616.322,A -85,B 0,C 180,E1 24068.91,E2 24068.91} C_VEL
LIN {X 0,Y 541.801,Z 740.4,A -85,B 0,C 180,E1 24066.961,E2 24066.961} C_VEL
LIN {X 0,Y 541.063,Z 763.545,A -85,B 0,C 180,E1 24066.411,E2 24066.411} C_VEL
LIN {X 0,Y 540.184,Z 785.15,A -85,B 0,C 180,E1 24065.717,E2 24065.717} C_VEL
LIN {X 0,Y 539.163,Z 806.346,A -85,B 0,C 180,E1 24064.835,E2 24064.835} C_VEL
LIN {X 0,Y 538.071,Z 826.207,A -85,B 0,C 180,E1 24063.838,E2 24063.838} C_VEL
LIN {X 0,Y 536.755,Z 847.21,A -85,B 0,C 180,E1 24062.573,E2 24062.573} C_VEL
LIN {X 0,Y 535.491,Z 867.378,A -85,B 0,C 180,E1 24061.148,E2 24061.148} C_VEL
LIN {X 0,Y 534.112,Z 887.247,A -85,B 0,C 180,E1 24059.497,E2 24059.497} C_VEL
LIN {X 0,Y 532.813,Z 906.767,A -85,B 0,C 180,E1 24057.616,E2 24057.616} C_VEL
LIN {X 0,Y 531.725,Z 923.639,A -85,B 0,C 180,E1 24055.748,E2 24055.748} C_VEL
LIN {X 0,Y 530.696,Z 939.975,A -85,B 0,C 180,E1 24053.662,E2 24053.662} C_VEL
LIN {X 0,Y 529.87,Z 954.91,A -85,B 0,C 180,E1 24051.476,E2 24051.476} C_VEL
LIN {X 0,Y 529.231,Z 967.714,A -85,B 0,C 180,E1 24049.309,E2 24049.309} C_VEL
LIN {X 0,Y 528.701,Z 980.047,A -85,B 0,C 180,E1 24046.879,E2 24046.879} C_VEL
LIN {X 0,Y 528.37,Z 989.979,A -85,B 0,C 180,E1 24044.58,E2 24044.58} C_VEL
LIN {X 0,Y 528.129,Z 998.691,A -85,B 0,C 180,E1 24042.134,E2 24042.134} C_VEL
LIN {X 0,Y 527.98,Z 1005.766,A -85,B 0,C 180,E1 24039.706,E2 24039.706} C_VEL
LIN {X 0,Y 527.919,Z 1010.835,A -85,B 0,C 180,E1 24037.403,E2 24037.403} C_VEL
LIN {X 0,Y 527.917,Z 1014.432,A -85,B 0,C 180,E1 24035.219,E2 24035.219} C_VEL
LIN {X 0,Y 527.908,Z 1017.054,A -85,B 0,C 180,E1 24032.609,E2 24032.609} C_VEL
LIN {X 0,Y 527.891,Z 1017.939,A -85,B 0,C 180,E1 24030.329,E2 24030.329} C_VEL
LIN {X 0,Y 527.915,Z 1017.326,A -85,B 0,C 180,E1 24027.833,E2 24027.833} C_VEL
LIN {X 0,Y 527.906,Z 1015.393,A -85,B 0,C 180,E1 24025.55,E2 24025.55} C_VEL
LIN {X 0,Y 527.909,Z 1011.674,A -85,B 0,C 180,E1 24023.041,E2 24023.041} C_VEL
LIN {X 0,Y 527.986,Z 1007.071,A -85,B 0,C 180,E1 24020.851,E2 24020.851} C_VEL
LIN {X 0,Y 528.099,Z 1000.129,A -85,B 0,C 180,E1 24018.316,E2 24018.316} C_VEL
LIN {X 0,Y 528.269,Z 992.537,A -85,B 0,C 180,E1 24016.095,E2 24016.095} C_VEL
LIN {X 0,Y 528.601,Z 982.415,A -85,B 0,C 180,E1 24013.634,E2 24013.634} C_VEL
LIN {X 0,Y 529.041,Z 971.429,A -85,B 0,C 180,E1 24011.378,E2 24011.378} C_VEL
LIN {X 0,Y 529.662,Z 958.488,A -85,B 0,C 180,E1 24009.102,E2 24009.102} C_VEL
LIN {X 0,Y 530.477,Z 944.053,A -85,B 0,C 180,E1 24006.895,E2 24006.895} C_VEL
LIN {X 0,Y 531.405,Z 928.331,A -85,B 0,C 180,E1 24004.825,E2 24004.825} C_VEL
LIN {X 0,Y 532.57,Z 910.163,A -85,B 0,C 180,E1 24002.741,E2 24002.741} C_VEL
LIN {X 0,Y 533.836,Z 891.954,A -85,B 0,C 180,E1 24000.925,E2 24000.925} C_VEL
LIN {X 0,Y 535.096,Z 872.566,A -85,B 0,C 180,E1 23999.264,E2 23999.264} C_VEL
LIN {X 0,Y 536.492,Z 851.803,A -85,B 0,C 180,E1 23997.733,E2 23997.733} C_VEL
LIN {X 0,Y 537.705,Z 831.899,A -85,B 0,C 180,E1 23996.483,E2 23996.483} C_VEL
LIN {X 0,Y 538.955,Z 810.356,A -85,B 0,C 180,E1 23995.352,E2 23995.352} C_VEL
LIN {X 0,Y 539.929,Z 791.105,A -85,B 0,C 180,E1 23994.516,E2 23994.516} C_VEL
LIN {X 0,Y 540.899,Z 767.519,A -85,B 0,C 180,E1 23993.702,E2 23993.702} C_VEL
LIN {X 0,Y 541.636,Z 746.146,A -85,B 0,C 180,E1 23993.156,E2 23993.156} C_VEL
LIN {X 0,Y 542.2,Z 714.391,A -85,B 0,C 180,E1 23992.611,E2 23992.611} C_VEL
LIN {X 0,Y 544.758,Z 503.857,A -85,B 0,C 180,E1 23989.32,E2 23989.32} C_VEL
LIN {X 0,Y 545.826,Z 408.074,A -85,B 0,C 180,E1 23987.771,E2 23987.771} C_VEL
LIN {X 0,Y 542.89,Z 394.737,A -85,B 0,C 180,E1 23987.255,E2 23987.255} C_VEL
LIN {X 0,Y 540.026,Z 390.002,A -85,B 0,C 180,E1 23986.843,E2 23986.843} C_VEL
LIN {X 0,Y 530.095,Z 369.079,A -85,B 0,C 180,E1 23984.107,E2 23984.107} C_VEL
LIN {X 0,Y 528.491,Z 365.462,A -85,B 0,C 180,E1 23983.571,E2 23983.571} C_VEL
LIN {X 0,Y 528.452,Z 365.22,A -85,B 0,C 180,E1 23981.18,E2 23981.18} C_VEL
LIN {X 0,Y 528.478,Z 365.22,A -85,B 0,C 180,E1 23977.806,E2 23977.806} C_VEL
LIN {X 0,Y 528.465,Z 365.199,A -85,B 0,C 180,E1 23974.583,E2 23974.583} C_VEL
LIN {X 0,Y 528.444,Z 365.206,A -85,B 0,C 180,E1 23971.226,E2 23971.226} C_VEL
LIN {X 0,Y 528.519,Z 365.214,A -85,B 0,C 180,E1 23967.947,E2 23967.947} C_VEL
LIN {X 0,Y 528.443,Z 365.22,A -85,B 0,C 180,E1 23964.598,E2 23964.598} C_VEL
LIN {X 0,Y 528.456,Z 365.216,A -85,B 0,C 180,E1 23961.144,E2 23961.144} C_VEL
LIN {X 0,Y 528.486,Z 365.217,A -85,B 0,C 180,E1 23957.909,E2 23957.909} C_VEL
LIN {X 0,Y 528.444,Z 365.214,A -85,B 0,C 180,E1 23954.575,E2 23954.575} C_VEL
LIN {X 0,Y 528.512,Z 365.213,A -85,B 0,C 180,E1 23951.347,E2 23951.347} C_VEL
LIN {X 0,Y 528.457,Z 365.213,A -85,B 0,C 180,E1 23948.048,E2 23948.048} C_VEL
LIN {X 0,Y 528.462,Z 365.216,A -85,B 0,C 180,E1 23944.557,E2 23944.557} C_VEL
LIN {X 0,Y 528.513,Z 365.213,A -85,B 0,C 180,E1 23941.3,E2 23941.3} C_VEL
LIN {X 0,Y 528.458,Z 365.214,A -85,B 0,C 180,E1 23938.048,E2 23938.048} C_VEL
LIN {X 0,Y 528.505,Z 365.214,A -85,B 0,C 180,E1 23934.681,E2 23934.681} C_VEL
LIN {X 0,Y 528.472,Z 365.211,A -85,B 0,C 180,E1 23931.513,E2 23931.513} C_VEL
LIN {X 0,Y 528.47,Z 365.213,A -85,B 0,C 180,E1 23927.987,E2 23927.987} C_VEL
LIN {X 0,Y 528.531,Z 365.211,A -85,B 0,C 180,E1 23924.642,E2 23924.642} C_VEL
LIN {X 0,Y 528.473,Z 365.211,A -85,B 0,C 180,E1 23921.352,E2 23921.352} C_VEL
LIN {X 0,Y 528.487,Z 365.211,A -85,B 0,C 180,E1 23917.883,E2 23917.883} C_VEL
LIN {X 0,Y 528.521,Z 365.211,A -85,B 0,C 180,E1 23914.568,E2 23914.568} C_VEL
LIN {X 0,Y 528.474,Z 365.209,A -85,B 0,C 180,E1 23911.277,E2 23911.277} C_VEL
LIN {X 0,Y 528.524,Z 365.21,A -85,B 0,C 180,E1 23907.933,E2 23907.933} C_VEL
LIN {X 0,Y 528.498,Z 365.212,A -85,B 0,C 180,E1 23904.618,E2 23904.618} C_VEL
LIN {X 0,Y 528.515,Z 365.209,A -85,B 0,C 180,E1 23901.607,E2 23901.607} C_VEL
LIN {X 0,Y 527.487,Z 365.338,A -85,B 0,C 180,E1 23900.772,E2 23900.772} C_VEL
LIN {X 0,Y 521.12,Z 366.14,A -85,B 0,C 180,E1 23898.426,E2 23898.426} C_VEL
LIN {X 0,Y 520.587,Z 366.201,A -85,B 0,C 180,E1 23897.815,E2 23897.815} C_VEL
LIN {X 0,Y 520.56,Z 366.204,A -85,B 0,C 180,E1 23894.396,E2 23894.396} C_VEL
LIN {X 0,Y 520.556,Z 366.2,A -85,B 0,C 180,E1 23890.911,E2 23890.911} C_VEL
LIN {X 0,Y 520.585,Z 366.199,A -85,B 0,C 180,E1 23887.5,E2 23887.5} C_VEL
LIN {X 0,Y 520.563,Z 366.187,A -85,B 0,C 180,E1 23884.109,E2 23884.109} C_VEL
LIN {X 0,Y 520.56,Z 366.201,A -85,B 0,C 180,E1 23880.592,E2 23880.592} C_VEL
LIN {X 0,Y 520.584,Z 366.203,A -85,B 0,C 180,E1 23877.196,E2 23877.196} C_VEL
LIN {X 0,Y 520.579,Z 366.196,A -85,B 0,C 180,E1 23873.662,E2 23873.662} C_VEL
LIN {X 0,Y 520.563,Z 366.193,A -85,B 0,C 180,E1 23870.222,E2 23870.222} C_VEL
LIN {X 0,Y 520.603,Z 366.365,A -85,B 0,C 180,E1 23867.142,E2 23867.142} C_VEL
LIN {X 0,Y 520.957,Z 367.797,A -85,B 0,C 180,E1 23866.936,E2 23866.936} C_VEL
LIN {X 0,Y 522.883,Z 370.845,A -85,B 0,C 180,E1 23866.66,E2 23866.66} C_VEL
LIN {X 0,Y 524.232,Z 372.387,A -85,B 0,C 180,E1 23866.484,E2 23866.484} C_VEL
LIN {X 0,Y 526.925,Z 376.348,A -85,B 0,C 180,E1 23866.12,E2 23866.12} C_VEL
LIN {X 0,Y 539.833,Z 395.13,A -85,B 0,C 180,E1 23864.462,E2 23864.462} C_VEL
LIN {X 0,Y 536.863,Z 606.497,A -85,B 0,C 180,E1 23861.085,E2 23861.085} C_VEL
LIN {X 0,Y 535.396,Z 711.308,A -85,B 0,C 180,E1 23859.418,E2 23859.418} C_VEL
LIN {X 0,Y 534.618,Z 733.828,A -85,B 0,C 180,E1 23858.876,E2 23858.876} C_VEL
LIN {X 0,Y 533.547,Z 757.047,A -85,B 0,C 180,E1 23858.11,E2 23858.11} C_VEL
LIN {X 0,Y 532.361,Z 778.92,A -85,B 0,C 180,E1 23857.171,E2 23857.171} C_VEL
LIN {X 0,Y 530.935,Z 801.302,A -85,B 0,C 180,E1 23855.996,E2 23855.996} C_VEL
LIN {X 0,Y 529.499,Z 822.488,A -85,B 0,C 180,E1 23854.654,E2 23854.654} C_VEL
LIN {X 0,Y 527.959,Z 843.355,A -85,B 0,C 180,E1 23853.091,E2 23853.091} C_VEL
LIN {X 0,Y 526.494,Z 863.158,A -85,B 0,C 180,E1 23851.357,E2 23851.357} C_VEL
LIN {X 0,Y 525.092,Z 881.333,A -85,B 0,C 180,E1 23849.506,E2 23849.506} C_VEL
LIN {X 0,Y 523.854,Z 898.64,A -85,B 0,C 180,E1 23847.481,E2 23847.481} C_VEL
LIN {X 0,Y 522.742,Z 915.315,A -85,B 0,C 180,E1 23845.228,E2 23845.228} C_VEL
LIN {X 0,Y 521.851,Z 929.883,A -85,B 0,C 180,E1 23842.953,E2 23842.953} C_VEL
LIN {X 0,Y 521.155,Z 942.746,A -85,B 0,C 180,E1 23840.611,E2 23840.611} C_VEL
LIN {X 0,Y 520.649,Z 954.366,A -85,B 0,C 180,E1 23838.139,E2 23838.139} C_VEL
LIN {X 0,Y 520.308,Z 963.687,A -85,B 0,C 180,E1 23835.758,E2 23835.758} C_VEL
LIN {X 0,Y 520.071,Z 971.926,A -85,B 0,C 180,E1 23833.223,E2 23833.223} C_VEL
LIN {X 0,Y 519.964,Z 978.124,A -85,B 0,C 180,E1 23830.8,E2 23830.8} C_VEL
LIN {X 0,Y 519.923,Z 983.013,A -85,B 0,C 180,E1 23828.258,E2 23828.258} C_VEL
LIN {X 0,Y 519.915,Z 986.211,A -85,B 0,C 180,E1 23825.695,E2 23825.695} C_VEL
LIN {X 0,Y 519.91,Z 987.779,A -85,B 0,C 180,E1 23823.129,E2 23823.129} C_VEL
LIN {X 0,Y 519.918,Z 987.774,A -85,B 0,C 180,E1 23820.757,E2 23820.757} C_VEL
LIN {X 0,Y 519.911,Z 986.197,A -85,B 0,C 180,E1 23818.199,E2 23818.199} C_VEL
LIN {X 0,Y 519.913,Z 983.091,A -85,B 0,C 180,E1 23815.701,E2 23815.701} C_VEL
LIN {X 0,Y 519.963,Z 978.16,A -85,B 0,C 180,E1 23813.126,E2 23813.126} C_VEL
LIN {X 0,Y 520.079,Z 972.138,A -85,B 0,C 180,E1 23810.762,E2 23810.762} C_VEL
LIN {X 0,Y 520.311,Z 963.77,A -85,B 0,C 180,E1 23808.176,E2 23808.176} C_VEL
LIN {X 0,Y 520.647,Z 954.284,A -85,B 0,C 180,E1 23805.752,E2 23805.752} C_VEL
LIN {X 0,Y 521.13,Z 943.002,A -85,B 0,C 180,E1 23803.348,E2 23803.348} C_VEL
LIN {X 0,Y 521.846,Z 929.792,A -85,B 0,C 180,E1 23800.941,E2 23800.941} C_VEL
LIN {X 0,Y 522.749,Z 915.208,A -85,B 0,C 180,E1 23798.666,E2 23798.666} C_VEL
LIN {X 0,Y 523.874,Z 898.496,A -85,B 0,C 180,E1 23796.411,E2 23796.411} C_VEL
LIN {X 0,Y 525.164,Z 880.388,A -85,B 0,C 180,E1 23794.302,E2 23794.302} C_VEL
LIN {X 0,Y 526.53,Z 862.666,A -85,B 0,C 180,E1 23792.508,E2 23792.508} C_VEL
LIN {X 0,Y 527.965,Z 843.304,A -85,B 0,C 180,E1 23790.816,E2 23790.816} C_VEL
LIN {X 0,Y 529.495,Z 822.508,A -85,B 0,C 180,E1 23789.258,E2 23789.258} C_VEL
LIN {X 0,Y 530.942,Z 801.216,A -85,B 0,C 180,E1 23787.909,E2 23787.909} C_VEL
LIN {X 0,Y 532.369,Z 778.791,A -85,B 0,C 180,E1 23786.732,E2 23786.732} C_VEL
LIN {X 0,Y 533.565,Z 756.737,A -85,B 0,C 180,E1 23785.788,E2 23785.788} C_VEL
LIN {X 0,Y 534.63,Z 733.52,A -85,B 0,C 180,E1 23785.025,E2 23785.025} C_VEL
LIN {X 0,Y 535.411,Z 710.84,A -85,B 0,C 180,E1 23784.482,E2 23784.482} C_VEL
LIN {X 0,Y 538.329,Z 499.573,A -85,B 0,C 180,E1 23781.13,E2 23781.13} C_VEL
LIN {X 0,Y 539.664,Z 394.918,A -85,B 0,C 180,E1 23779.427,E2 23779.427} C_VEL
LIN {X 0,Y 529.75,Z 380.47,A -85,B 0,C 180,E1 23778.16,E2 23778.16} C_VEL
LIN {X 0,Y 526.436,Z 375.772,A -85,B 0,C 180,E1 23777.72,E2 23777.72} C_VEL
LIN {X 0,Y 523.596,Z 371.501,A -85,B 0,C 180,E1 23777.332,E2 23777.332} C_VEL
LIN {X 0,Y 521.284,Z 368.66,A -85,B 0,C 180,E1 23777.023,E2 23777.023} C_VEL
LIN {X 0,Y 520.666,Z 366.852,A -85,B 0,C 180,E1 23776.857,E2 23776.857} C_VEL
LIN {X 0,Y 520.569,Z 366.196,A -85,B 0,C 180,E1 23776.515,E2 23776.515} C_VEL
LIN {X 0,Y 520.565,Z 366.203,A -85,B 0,C 180,E1 23772.987,E2 23772.987} C_VEL
LIN {X 0,Y 520.581,Z 366.198,A -85,B 0,C 180,E1 23769.508,E2 23769.508} C_VEL
LIN {X 0,Y 520.58,Z 366.201,A -85,B 0,C 180,E1 23765.954,E2 23765.954} C_VEL
LIN {X 0,Y 520.574,Z 366.199,A -85,B 0,C 180,E1 23762.532,E2 23762.532} C_VEL
LIN {X 0,Y 520.584,Z 366.199,A -85,B 0,C 180,E1 23759.01,E2 23759.01} C_VEL
LIN {X 0,Y 520.562,Z 366.202,A -85,B 0,C 180,E1 23755.484,E2 23755.484} C_VEL
LIN {X 0,Y 520.587,Z 366.203,A -85,B 0,C 180,E1 23752.052,E2 23752.052} C_VEL
LIN {X 0,Y 520.584,Z 366.199,A -85,B 0,C 180,E1 23748.591,E2 23748.591} C_VEL
LIN {X 0,Y 520.547,Z 366.204,A -85,B 0,C 180,E1 23745.199,E2 23745.199} C_VEL
LIN {X 0,Y 520.574,Z 366.204,A -85,B 0,C 180,E1 23741.756,E2 23741.756} C_VEL
LIN {X 0,Y 520.575,Z 366.198,A -85,B 0,C 180,E1 23738.361,E2 23738.361} C_VEL
LIN {X 0,Y 520.531,Z 366.206,A -85,B 0,C 180,E1 23735.003,E2 23735.003} C_VEL
LIN {X 0,Y 520.565,Z 366.202,A -85,B 0,C 180,E1 23731.608,E2 23731.608} C_VEL
LIN {X 0,Y 520.537,Z 366.204,A -85,B 0,C 180,E1 23728.374,E2 23728.374} C_VEL
LIN {X 0,Y 520.513,Z 366.21,A -85,B 0,C 180,E1 23724.918,E2 23724.918} C_VEL
LIN {X 0,Y 520.57,Z 366.201,A -85,B 0,C 180,E1 23721.598,E2 23721.598} C_VEL
LIN {X 0,Y 520.51,Z 366.214,A -85,B 0,C 180,E1 23718.346,E2 23718.346} C_VEL
LIN {X 0,Y 520.572,Z 366.491,A -85,B 0,C 180,E1 23717.163,E2 23717.163} C_VEL
LIN {X 0,Y 521.828,Z 369.724,A -85,B 0,C 180,E1 23716.69,E2 23716.69} C_VEL
LIN {X 0,Y 526.712,Z 379.739,A -85,B 0,C 180,E1 23715.307,E2 23715.307} C_VEL
LIN {X 0,Y 532.126,Z 390.843,A -85,B 0,C 180,E1 23713.884,E2 23713.884} C_VEL
LIN {X 0,Y 537.873,Z 400.137,A -85,B 0,C 180,E1 23713.136,E2 23713.136} C_VEL
LIN {X 0,Y 540.012,Z 411.685,A -85,B 0,C 180,E1 23712.723,E2 23712.723} C_VEL
LIN {X 0,Y 537.107,Z 618.331,A -85,B 0,C 180,E1 23709.416,E2 23709.416} C_VEL
LIN {X 0,Y 535.403,Z 740.41,A -85,B 0,C 180,E1 23707.478,E2 23707.478} C_VEL
LIN {X 0,Y 534.605,Z 763.413,A -85,B 0,C 180,E1 23706.927,E2 23706.927} C_VEL
LIN {X 0,Y 533.65,Z 784.722,A -85,B 0,C 180,E1 23706.239,E2 23706.239} C_VEL
LIN {X 0,Y 532.492,Z 806.343,A -85,B 0,C 180,E1 23705.336,E2 23705.336} C_VEL
LIN {X 0,Y 531.277,Z 826.534,A -85,B 0,C 180,E1 23704.311,E2 23704.311} C_VEL
LIN {X 0,Y 529.773,Z 848.106,A -85,B 0,C 180,E1 23702.993,E2 23702.993} C_VEL
LIN {X 0,Y 528.375,Z 868.158,A -85,B 0,C 180,E1 23701.552,E2 23701.552} C_VEL
LIN {X 0,Y 526.897,Z 887.245,A -85,B 0,C 180,E1 23699.942,E2 23699.942} C_VEL
LIN {X 0,Y 525.42,Z 907.141,A -85,B 0,C 180,E1 23697.997,E2 23697.997} C_VEL
LIN {X 0,Y 524.213,Z 923.638,A -85,B 0,C 180,E1 23696.145,E2 23696.145} C_VEL
LIN {X 0,Y 523.075,Z 939.974,A -85,B 0,C 180,E1 23694.029,E2 23694.029} C_VEL
LIN {X 0,Y 522.123,Z 955.234,A -85,B 0,C 180,E1 23691.758,E2 23691.758} C_VEL
LIN {X 0,Y 521.411,Z 967.712,A -85,B 0,C 180,E1 23689.611,E2 23689.611} C_VEL
LIN {X 0,Y 520.803,Z 980.313,A -85,B 0,C 180,E1 23687.085,E2 23687.085} C_VEL
LIN {X 0,Y 520.424,Z 990.437,A -85,B 0,C 180,E1 23684.694,E2 23684.694} C_VEL
LIN {X 0,Y 520.153,Z 999.048,A -85,B 0,C 180,E1 23682.21,E2 23682.21} C_VEL
LIN {X 0,Y 519.989,Z 1006.035,A -85,B 0,C 180,E1 23679.745,E2 23679.745} C_VEL
LIN {X 0,Y 519.922,Z 1011.042,A -85,B 0,C 180,E1 23677.406,E2 23677.406} C_VEL
LIN {X 0,Y 519.914,Z 1014.75,A -85,B 0,C 180,E1 23675.078,E2 23675.078} C_VEL
LIN {X 0,Y 519.911,Z 1017.121,A -85,B 0,C 180,E1 23672.538,E2 23672.538} C_VEL
LIN {X 0,Y 519.905,Z 1017.983,A -85,B 0,C 180,E1 23670.114,E2 23670.114} C_VEL
LIN {X 0,Y 519.914,Z 1017.259,A -85,B 0,C 180,E1 23667.689,E2 23667.689} C_VEL
LIN {X 0,Y 519.905,Z 1015.165,A -85,B 0,C 180,E1 23665.26,E2 23665.26} C_VEL
LIN {X 0,Y 519.912,Z 1011.468,A -85,B 0,C 180,E1 23662.823,E2 23662.823} C_VEL
LIN {X 0,Y 519.989,Z 1007.071,A -85,B 0,C 180,E1 23660.709,E2 23660.709} C_VEL
LIN {X 0,Y 520.134,Z 999.968,A -85,B 0,C 180,E1 23658.083,E2 23658.083} C_VEL
